C03643=1229.228,50.158,-44.225,-178.947,5.404,148.624
C03644=1229.233,49.908,-44.209,-178.950,5.403,148.624
C03645=1229.238,49.659,-44.193,-178.952,5.403,148.625
C03646=1229.242,49.409,-44.176,-178.955,5.402,148.626
C03647=1229.248,49.160,-44.159,-178.958,5.401,148.626
C03648=1229.253,48.911,-44.143,-178.960,5.401,148.627
C03649=1229.257,48.661,-44.126,-178.962,5.400,148.628
C03650=1229.263,48.412,-44.111,-178.965,5.399,148.628
C03651=1229.267,48.162,-44.094,-178.968,5.399,148.629
C03652=1229.272,47.913,-44.077,-178.970,5.398,148.630
C03653=1229.277,47.664,-44.060,-178.972,5.398,148.630
C03654=1229.282,47.414,-44.044,-178.975,5.398,148.631
C03655=1229.287,47.165,-44.028,-178.978,5.397,148.632
C03656=1229.292,46.915,-44.011,-178.980,5.397,148.632
C03657=1229.296,46.666,-43.995,-178.983,5.396,148.633
C03658=1229.302,46.416,-43.979,-178.986,5.396,148.634
C03659=1229.307,46.167,-43.962,-178.988,5.395,148.634
C03660=1229.312,45.918,-43.946,-178.990,5.394,148.635
C03661=1229.316,45.668,-43.929,-178.993,5.394,148.635
C03662=1229.322,45.419,-43.913,-178.996,5.393,148.636
C03663=1229.326,45.170,-43.897,-178.998,5.392,148.637
C03664=1229.331,44.920,-43.880,-179.000,5.393,148.637
C03665=1229.337,44.670,-43.864,-179.003,5.392,148.638
C03666=1229.341,44.421,-43.847,-179.006,5.392,148.639
C03667=1229.346,44.172,-43.831,-179.008,5.391,148.639
C03668=1229.351,43.922,-43.815,-179.011,5.390,148.640
C03669=1229.356,43.673,-43.799,-179.013,5.389,148.641
C03670=1229.361,43.423,-43.783,-179.016,5.389,148.641
C03671=1229.366,43.174,-43.766,-179.018,5.388,148.642
C03672=1229.371,42.925,-43.750,-179.021,5.388,148.643
C03673=1229.376,42.675,-43.734,-179.023,5.388,148.643
C03674=1229.380,42.426,-43.717,-179.026,5.387,148.644
C03675=1229.386,42.177,-43.702,-179.028,5.387,148.645
C03676=1229.390,41.927,-43.685,-179.031,5.386,148.645
C03677=1229.395,41.678,-43.669,-179.034,5.386,148.646
C03678=1229.401,41.428,-43.652,-179.036,5.385,148.647
C03679=1229.406,41.179,-43.636,-179.039,5.385,148.647
C03680=1229.411,40.929,-43.620,-179.041,5.384,148.648
C03681=1229.416,40.680,-43.604,-179.043,5.384,148.648
C03682=1229.421,40.430,-43.588,-179.046,5.383,148.649
C03683=1229.426,40.181,-43.572,-179.048,5.383,148.650
C03684=1229.430,39.931,-43.556,-179.051,5.382,148.650
C03685=1229.436,39.682,-43.539,-179.054,5.382,148.651
C03686=1229.440,39.432,-43.523,-179.056,5.381,148.652
C03687=1229.445,39.184,-43.507,-179.059,5.381,148.652
C03688=1229.450,38.933,-43.491,-179.062,5.380,148.653
C03689=1229.455,38.685,-43.475,-179.064,5.380,148.654
C03690=1229.460,38.435,-43.459,-179.066,5.380,148.654
C03691=1229.465,38.186,-43.442,-179.069,5.379,148.655
C03692=1229.470,37.936,-43.427,-179.072,5.379,148.656
C03693=1229.475,37.686,-43.411,-179.074,5.378,148.656
C03694=1229.480,37.438,-43.395,-179.076,5.377,148.657
C03695=1229.484,37.188,-43.379,-179.079,5.377,148.658
C03696=1229.490,36.939,-43.363,-179.082,5.376,148.658
C03697=1229.494,36.689,-43.347,-179.084,5.376,148.659
C03698=1229.500,36.439,-43.331,-179.086,5.376,148.660
C03699=1229.504,36.190,-43.315,-179.089,5.375,148.660
C03700=1229.510,35.941,-43.299,-179.092,5.375,148.661
C03701=1229.515,35.692,-43.283,-179.094,5.374,148.662
C03702=1229.519,35.442,-43.267,-179.097,5.374,148.662
C03703=1229.525,35.192,-43.251,-179.100,5.373,148.663
C03704=1229.529,34.943,-43.235,-179.102,5.373,148.664
C03705=1229.535,34.693,-43.219,-179.104,5.373,148.664
C03706=1229.539,34.444,-43.204,-179.107,5.372,148.665
C03707=1229.544,34.195,-43.187,-179.110,5.372,148.666
C03708=1229.549,33.945,-43.172,-179.112,5.371,148.666
C03709=1229.554,33.695,-43.156,-179.114,5.370,148.667
C03710=1229.559,33.446,-43.140,-179.117,5.370,148.668
C03711=1229.564,33.197,-43.124,-179.119,5.370,148.668
C03712=1229.569,32.947,-43.108,-179.122,5.369,148.669
C03713=1229.574,32.698,-43.093,-179.124,5.369,148.670
C03714=1229.578,32.448,-43.076,-179.127,5.368,148.670
C03715=1229.584,32.199,-43.061,-179.130,5.368,148.671
C03716=1229.589,31.950,-43.045,-179.132,5.367,148.672
C03717=1229.594,31.700,-43.029,-179.134,5.367,148.672
C03718=1229.599,31.451,-43.013,-179.137,5.367,148.673
C03719=1229.604,31.202,-42.998,-179.140,5.366,148.674
C03720=1229.608,30.952,-42.982,-179.142,5.366,148.674
C03721=1229.614,30.702,-42.966,-179.145,5.365,148.675
C03722=1229.619,30.453,-42.951,-179.148,5.365,148.676
C03723=1229.624,30.203,-42.934,-179.150,5.365,148.676
C03724=1229.629,29.934,-42.918,-179.152,5.364,148.677
C03725=1229.634,29.666,-42.901,-179.155,5.364,148.678
C03726=1229.640,29.398,-42.884,-179.158,5.363,148.678
C03727=1229.646,29.129,-42.867,-179.160,5.363,148.679
C03728=1229.650,28.879,-42.851,-179.163,5.362,148.680
C03729=1229.655,28.630,-42.836,-179.165,5.361,148.680
C03730=1229.660,28.381,-42.820,-179.168,5.361,148.681
C03731=1229.665,28.131,-42.804,-179.171,5.360,148.682
C03732=1229.670,27.882,-42.789,-179.173,5.361,148.682
C03733=1229.675,27.632,-42.774,-179.175,5.360,148.683
C03734=1229.680,27.382,-42.758,-179.178,5.360,148.684
C03735=1229.685,27.133,-42.742,-179.181,5.359,148.685
C03736=1229.690,26.884,-42.727,-179.183,5.358,148.685
C03737=1229.695,26.634,-42.711,-179.186,5.358,148.686
C03738=1229.700,26.384,-42.696,-179.188,5.358,148.687
C03739=1229.705,26.135,-42.680,-179.191,5.358,148.687
C03740=1229.710,25.886,-42.665,-179.193,5.357,148.688
C03741=1229.715,25.636,-42.649,-179.196,5.357,148.689
C03742=1229.720,25.387,-42.633,-179.199,5.356,148.689
C03743=1229.724,25.138,-42.618,-179.201,5.356,148.690
C03744=1229.730,24.888,-42.602,-179.203,5.356,148.691
C03745=1229.735,24.638,-42.586,-179.206,5.355,148.691
C03746=1229.739,24.389,-42.571,-179.208,5.354,148.692
C03747=1229.745,24.140,-42.556,-179.211,5.354,148.692
C03748=1229.750,23.890,-42.540,-179.214,5.353,148.693
C03749=1229.754,23.641,-42.525,-179.216,5.353,148.694
C03750=1229.760,23.391,-42.510,-179.218,5.353,148.694
C03751=1229.764,23.142,-42.495,-179.221,5.352,148.695
C03752=1229.770,22.892,-42.479,-179.224,5.352,148.696
C03753=1229.775,22.642,-42.463,-179.226,5.351,148.697
C03754=1229.779,22.393,-42.448,-179.228,5.351,148.697
C03755=1229.785,22.144,-42.433,-179.231,5.351,148.698
C03756=1229.790,21.894,-42.417,-179.234,5.350,148.699
C03757=1229.795,21.645,-42.402,-179.236,5.350,148.699
C03758=1229.799,21.395,-42.386,-179.239,5.349,148.700
C03759=1229.804,21.146,-42.371,-179.241,5.350,148.701
C03760=1229.809,20.896,-42.356,-179.244,5.349,148.701
C03761=1229.814,20.647,-42.341,-179.246,5.348,148.702
C03762=1229.819,20.398,-42.325,-179.249,5.348,148.703
C03763=1229.825,20.147,-42.310,-179.251,5.347,148.703
C03764=1229.829,19.898,-42.295,-179.254,5.348,148.704
C03765=1229.835,19.649,-42.279,-179.256,5.347,148.705
C03766=1229.839,19.400,-42.264,-179.259,5.347,148.705
C03767=1229.845,19.150,-42.249,-179.261,5.346,148.706
C03768=1229.849,18.900,-42.233,-179.264,5.346,148.707
C03769=1229.854,18.650,-42.218,-179.266,5.346,148.707
C03770=1229.859,18.401,-42.203,-179.269,5.345,148.708
C03771=1229.864,18.152,-42.188,-179.272,5.345,148.709
C03772=1229.869,17.903,-42.173,-179.274,5.344,148.709
C03773=1229.874,17.653,-42.157,-179.276,5.344,148.710
C03774=1229.879,17.403,-42.143,-179.279,5.344,148.711
C03775=1229.884,17.154,-42.127,-179.282,5.343,148.712
C03776=1229.889,16.905,-42.112,-179.284,5.343,148.712
C03777=1229.894,16.655,-42.096,-179.287,5.342,148.713
C03778=1229.899,16.405,-42.082,-179.289,5.343,148.714
C03779=1229.905,16.156,-42.066,-179.292,5.342,148.714
C03780=1229.909,15.907,-42.051,-179.294,5.341,148.715
C03781=1229.915,15.658,-42.036,-179.297,5.341,148.716
C03782=1229.919,15.407,-42.021,-179.299,5.341,148.716
C03783=1229.924,15.158,-42.006,-179.301,5.340,148.717
C03784=1229.929,14.909,-41.991,-179.304,5.340,148.717
C03785=1229.934,14.659,-41.976,-179.306,5.339,148.718
C03786=1229.939,14.410,-41.961,-179.309,5.339,148.719
C03787=1229.944,14.160,-41.946,-179.311,5.339,148.720
C03788=1229.950,13.910,-41.931,-179.314,5.338,148.720
C03789=1229.954,13.661,-41.916,-179.316,5.338,148.721
C03790=1229.960,13.412,-41.900,-179.319,5.337,148.722
C03791=1229.964,13.162,-41.886,-179.321,5.338,148.722
C03792=1229.969,12.912,-41.871,-179.324,5.337,148.723
C03793=1229.974,12.663,-41.855,-179.326,5.336,148.724
C03794=1229.979,12.413,-41.841,-179.329,5.336,148.724
C03795=1229.984,12.164,-41.825,-179.331,5.336,148.725
C03796=1229.989,11.915,-41.810,-179.334,5.336,148.726
C03797=1229.994,11.665,-41.796,-179.336,5.335,148.726
C03798=1229.999,11.416,-41.780,-179.339,5.335,148.727
C03799=1230.004,11.166,-41.766,-179.341,5.335,148.728
C03800=1230.009,10.917,-41.751,-179.344,5.334,148.728
C03801=1230.015,10.667,-41.736,-179.346,5.334,148.729
C03802=1230.019,10.418,-41.721,-179.349,5.333,148.730
C03803=1230.024,10.169,-41.706,-179.351,5.334,148.730
C03804=1230.030,9.919,-41.691,-179.354,5.333,148.731
C03805=1230.034,9.670,-41.676,-179.356,5.332,148.732
C03806=1230.039,9.420,-41.662,-179.359,5.332,148.733
C03807=1230.045,9.170,-41.647,-179.362,5.331,148.733
C03808=1230.050,8.921,-41.632,-179.364,5.332,148.734
C03809=1230.054,8.672,-41.617,-179.367,5.331,148.735
C03810=1230.060,8.422,-41.602,-179.369,5.331,148.735
C03811=1230.064,8.172,-41.587,-179.372,5.330,148.736
C03812=1230.069,7.922,-41.573,-179.374,5.330,148.737
C03813=1230.074,7.673,-41.558,-179.377,5.330,148.737
C03814=1230.079,7.423,-41.543,-179.379,5.329,148.738
C03815=1230.084,7.174,-41.528,-179.381,5.330,148.739
C03816=1230.089,6.924,-41.514,-179.384,5.329,148.739
C03817=1230.094,6.675,-41.499,-179.387,5.329,148.740
C03818=1230.099,6.425,-41.484,-179.389,5.328,148.741
C03819=1230.104,6.175,-41.469,-179.391,5.328,148.741
C03820=1230.109,5.926,-41.455,-179.394,5.328,148.742
C03821=1230.114,5.677,-41.440,-179.397,5.327,148.743
C03822=1230.120,5.428,-41.425,-179.399,5.327,148.744
C03823=1230.125,5.178,-41.411,-179.401,5.327,148.744
C03824=1230.130,4.928,-41.396,-179.404,5.326,148.745
C03825=1230.134,4.679,-41.381,-179.407,5.326,148.746
C03826=1230.140,4.429,-41.367,-179.409,5.325,148.746
C03827=1230.145,4.180,-41.352,-179.411,5.326,148.747
C03828=1230.150,3.911,-41.337,-179.414,5.325,148.748
C03829=1230.155,3.642,-41.321,-179.417,5.325,148.749
C03830=1230.161,3.373,-41.305,-179.420,5.324,148.749
C03831=1230.166,3.104,-41.289,-179.422,5.324,148.750
C03832=1230.171,2.854,-41.275,-179.425,5.323,148.751
C03833=1230.176,2.605,-41.260,-179.427,5.324,148.751
C03834=1230.181,2.356,-41.245,-179.430,5.323,148.752
C03835=1230.187,2.106,-41.230,-179.432,5.323,148.753
C03836=1230.191,1.857,-41.215,-179.435,5.323,148.753
C03837=1230.196,1.607,-41.201,-179.437,5.322,148.754
C03838=1230.201,1.357,-41.187,-179.440,5.322,148.755
C03839=1230.207,1.108,-41.173,-179.443,5.321,148.755
C03840=1230.211,0.859,-41.158,-179.445,5.322,148.756
C03841=1230.216,0.609,-41.144,-179.447,5.321,148.757
C03842=1230.222,0.359,-41.129,-179.450,5.321,148.758
C03843=1230.227,0.110,-41.115,-179.453,5.320,148.758
C03844=1230.232,-0.139,-41.100,-179.455,5.320,148.759
C03845=1230.237,-0.389,-41.085,-179.457,5.320,148.760
C03846=1230.241,-0.639,-41.071,-179.460,5.319,148.760
C03847=1230.246,-0.889,-41.057,-179.462,5.320,148.761
C03848=1230.252,-1.138,-41.043,-179.465,5.319,148.762
C03849=1230.257,-1.387,-41.028,-179.467,5.318,148.762
C03850=1230.262,-1.636,-41.014,-179.470,5.318,148.763
C03851=1230.267,-1.886,-40.999,-179.472,5.318,148.764
C03852=1230.272,-2.136,-40.985,-179.475,5.318,148.764
C03853=1230.276,-2.386,-40.971,-179.477,5.317,148.765
C03854=1230.282,-2.636,-40.956,-179.479,5.317,148.766
C03855=1230.287,-2.885,-40.941,-179.482,5.317,148.766
C03856=1230.292,-3.134,-40.927,-179.485,5.317,148.767
C03857=1230.297,-3.383,-40.913,-179.487,5.317,148.768
C03858=1230.302,-3.633,-40.898,-179.490,5.317,148.769
C03859=1230.307,-3.883,-40.884,-179.493,5.316,148.769
C03860=1230.312,-4.133,-40.870,-179.495,5.316,148.770
C03861=1230.317,-4.382,-40.856,-179.497,5.316,148.771
C03862=1230.323,-4.631,-40.842,-179.500,5.315,148.772
C03863=1230.327,-4.880,-40.827,-179.503,5.315,148.772
C03864=1230.332,-5.130,-40.812,-179.505,5.315,148.773
C03865=1230.337,-5.380,-40.798,-179.507,5.315,148.774
C03866=1230.342,-5.629,-40.784,-179.510,5.314,148.774
C03867=1230.347,-5.879,-40.770,-179.513,5.313,148.775
C03868=1230.353,-6.128,-40.756,-179.515,5.314,148.776
C03869=1230.358,-6.378,-40.741,-179.517,5.313,148.776
C03870=1230.363,-6.628,-40.727,-179.520,5.313,148.777
C03871=1230.368,-6.877,-40.713,-179.522,5.313,148.778
C03872=1230.373,-7.127,-40.699,-179.525,5.312,148.778
C03873=1230.378,-7.376,-40.685,-179.528,5.312,148.779
C03874=1230.382,-7.625,-40.671,-179.530,5.312,148.780
C03875=1230.387,-7.875,-40.657,-179.532,5.312,148.781
C03876=1230.392,-8.125,-40.642,-179.535,5.311,148.781
C03877=1230.397,-8.375,-40.628,-179.537,5.312,148.782
C03878=1230.403,-8.624,-40.614,-179.540,5.311,148.783
C03879=1230.408,-8.873,-40.600,-179.542,5.310,148.783
C03880=1230.413,-9.123,-40.586,-179.545,5.310,148.784
C03881=1230.418,-9.373,-40.571,-179.547,5.310,148.785
C03882=1230.423,-9.622,-40.557,-179.550,5.310,148.785
C03883=1230.428,-9.871,-40.543,-179.552,5.309,148.786
C03884=1230.433,-10.121,-40.529,-179.554,5.309,148.787
C03885=1230.438,-10.371,-40.515,-179.557,5.309,148.787
C03886=1230.443,-10.620,-40.502,-179.560,5.308,148.788
C03887=1230.448,-10.870,-40.488,-179.562,5.309,148.789
C03888=1230.453,-11.120,-40.473,-179.564,5.308,148.790
C03889=1230.458,-11.369,-40.459,-179.567,5.308,148.790
C03890=1230.464,-11.618,-40.445,-179.569,5.308,148.791
C03891=1230.469,-11.868,-40.431,-179.572,5.307,148.792
C03892=1230.473,-12.118,-40.417,-179.575,5.307,148.792
C03893=1230.478,-12.367,-40.403,-179.577,5.307,148.793
C03894=1230.484,-12.617,-40.390,-179.579,5.307,148.794
C03895=1230.489,-12.866,-40.376,-179.582,5.306,148.794
C03896=1230.493,-13.116,-40.361,-179.584,5.307,148.795
C03897=1230.499,-13.365,-40.347,-179.587,5.306,148.796
C03898=1230.504,-13.615,-40.333,-179.589,5.306,148.796
C03899=1230.508,-13.864,-40.319,-179.591,5.306,148.797
C03900=1230.513,-14.115,-40.306,-179.595,5.306,148.798
C03901=1230.519,-14.364,-40.292,-179.597,5.305,148.799
C03902=1230.524,-14.613,-40.278,-179.599,5.305,148.799
C03903=1230.529,-14.863,-40.263,-179.602,5.305,148.800
C03904=1230.534,-15.112,-40.251,-179.605,5.304,148.801
C03905=1230.539,-15.362,-40.237,-179.607,5.305,148.802
C03906=1230.544,-15.612,-40.222,-179.609,5.304,148.802
C03907=1230.550,-15.861,-40.208,-179.612,5.304,148.803
C03908=1230.554,-16.111,-40.195,-179.614,5.304,148.804
C03909=1230.559,-16.361,-40.181,-179.617,5.303,148.804
C03910=1230.565,-16.610,-40.167,-179.619,5.303,148.805
C03911=1230.569,-16.859,-40.153,-179.621,5.303,148.806
C03912=1230.574,-17.109,-40.140,-179.624,5.303,148.806
C03913=1230.580,-17.358,-40.126,-179.627,5.302,148.807
C03914=1230.585,-17.608,-40.112,-179.629,5.303,148.808
C03915=1230.590,-17.858,-40.098,-179.632,5.302,148.808
C03916=1230.595,-18.107,-40.085,-179.634,5.302,148.809
C03917=1230.600,-18.357,-40.071,-179.636,5.302,148.810
C03918=1230.605,-18.607,-40.057,-179.639,5.301,148.811
C03919=1230.610,-18.856,-40.043,-179.642,5.301,148.811
C03920=1230.615,-19.105,-40.029,-179.644,5.301,148.812
C03921=1230.620,-19.355,-40.016,-179.646,5.301,148.813
C03922=1230.625,-19.605,-40.002,-179.649,5.300,148.813
C03923=1230.630,-19.854,-39.988,-179.651,5.300,148.814
C03924=1230.635,-20.104,-39.975,-179.654,5.300,148.815
C03925=1230.640,-20.354,-39.961,-179.656,5.299,148.815
C03926=1230.645,-20.602,-39.948,-179.658,5.300,148.816
C03927=1230.651,-20.853,-39.934,-179.661,5.299,148.817
C03928=1230.655,-21.102,-39.920,-179.664,5.299,148.818
C03929=1230.661,-21.352,-39.907,-179.666,5.299,148.818
C03930=1230.666,-21.601,-39.893,-179.669,5.299,148.819
C03931=1230.671,-21.851,-39.880,-179.672,5.298,148.820
C03932=1230.676,-22.120,-39.865,-179.674,5.299,148.821
C03933=1230.682,-22.389,-39.850,-179.676,5.298,148.821
C03934=1230.687,-22.659,-39.835,-179.679,5.298,148.822
C03935=1230.693,-22.928,-39.821,-179.682,5.297,148.823
C03936=1230.698,-23.178,-39.808,-179.684,5.298,148.824
C03937=1230.702,-23.427,-39.793,-179.687,5.297,148.824
C03938=1230.708,-23.677,-39.780,-179.690,5.297,148.825
C03939=1230.713,-23.926,-39.766,-179.692,5.297,148.826
C03940=1230.718,-24.176,-39.753,-179.694,5.297,148.826
C03941=1230.723,-24.425,-39.740,-179.696,5.297,148.827
C03942=1230.729,-24.675,-39.726,-179.699,5.296,148.828
C03943=1230.733,-24.924,-39.713,-179.702,5.296,148.828
C03944=1230.738,-25.175,-39.699,-179.704,5.296,148.829
C03945=1230.744,-25.424,-39.685,-179.706,5.296,148.830
C03946=1230.748,-25.674,-39.672,-179.709,5.295,148.831
C03947=1230.754,-25.923,-39.658,-179.711,5.295,148.831
C03948=1230.758,-26.173,-39.645,-179.714,5.295,148.832
C03949=1230.764,-26.422,-39.631,-179.717,5.294,148.833
C03950=1230.768,-26.672,-39.619,-179.719,5.295,148.833
C03951=1230.774,-26.921,-39.605,-179.721,5.294,148.834
C03952=1230.778,-27.171,-39.592,-179.723,5.295,148.835
C03953=1230.784,-27.420,-39.578,-179.726,5.294,148.835
C03954=1230.788,-27.670,-39.565,-179.729,5.293,148.836
C03955=1230.794,-27.920,-39.552,-179.731,5.294,148.837
C03956=1230.799,-28.170,-39.539,-179.733,5.293,148.837
C03957=1230.804,-28.419,-39.525,-179.736,5.293,148.838
C03958=1230.809,-28.669,-39.512,-179.739,5.293,148.839
C03959=1230.815,-28.918,-39.499,-179.741,5.293,148.840
C03960=1230.819,-29.168,-39.485,-179.743,5.293,148.841
C03961=1230.825,-29.417,-39.472,-179.746,5.293,148.841
C03962=1230.829,-29.667,-39.458,-179.749,5.292,148.842
C03963=1230.835,-29.916,-39.445,-179.751,5.293,148.843
C03964=1230.839,-30.166,-39.432,-179.753,5.292,148.843
C03965=1230.845,-30.416,-39.419,-179.756,5.292,148.844
C03966=1230.849,-30.665,-39.405,-179.758,5.292,148.845
C03967=1230.855,-30.915,-39.392,-179.761,5.291,148.845
C03968=1230.860,-31.165,-39.379,-179.763,5.292,148.846
C03969=1230.865,-31.414,-39.365,-179.766,5.291,148.847
C03970=1230.871,-31.663,-39.352,-179.768,5.291,148.847
C03971=1230.875,-31.913,-39.339,-179.770,5.291,148.848
C03972=1230.881,-32.163,-39.326,-179.773,5.291,148.849
C03973=1230.885,-32.412,-39.312,-179.776,5.290,148.850
C03974=1230.891,-32.662,-39.299,-179.778,5.290,148.850
C03975=1230.896,-32.912,-39.286,-179.780,5.290,148.851
C03976=1230.901,-33.161,-39.274,-179.783,5.290,148.852
C03977=1230.906,-33.411,-39.259,-179.785,5.290,148.852
C03978=1230.911,-33.660,-39.247,-179.788,5.289,148.853
C03979=1230.917,-33.910,-39.234,-179.790,5.289,148.854
C03980=1230.921,-34.160,-39.221,-179.793,5.289,148.854
C03981=1230.926,-34.409,-39.208,-179.795,5.289,148.855
C03982=1230.931,-34.659,-39.194,-179.797,5.289,148.856
C03983=1230.936,-34.908,-39.181,-179.801,5.289,148.857
C03984=1230.942,-35.158,-39.168,-179.803,5.289,148.858
C03985=1230.947,-35.408,-39.155,-179.805,5.288,148.858
C03986=1230.952,-35.657,-39.142,-179.807,5.289,148.859
C03987=1230.957,-35.907,-39.128,-179.810,5.288,148.860
C03988=1230.962,-36.156,-39.115,-179.813,5.288,148.860
C03989=1230.967,-36.406,-39.103,-179.815,5.288,148.861
C03990=1230.972,-36.656,-39.089,-179.817,5.288,148.862
C03991=1230.977,-36.905,-39.077,-179.820,5.287,148.862
C03992=1230.983,-37.155,-39.064,-179.822,5.287,148.863
C03993=1230.988,-37.405,-39.051,-179.825,5.287,148.864
C03994=1230.993,-37.654,-39.038,-179.827,5.287,148.865
C03995=1230.997,-37.904,-39.025,-179.830,5.287,148.865
C03996=1231.003,-38.153,-39.011,-179.832,5.286,148.866
C03997=1231.008,-38.403,-38.998,-179.834,5.287,148.867
C03998=1231.013,-38.653,-38.986,-179.837,5.286,148.867
C03999=1231.018,-38.902,-38.973,-179.839,5.286,148.868
C04000=1231.024,-39.152,-38.960,-179.842,5.286,148.869
C04001=1231.028,-39.402,-38.947,-179.844,5.285,148.869
C04002=1231.033,-39.651,-38.934,-179.846,5.286,148.870
C04003=1231.038,-39.900,-38.922,-179.849,5.285,148.871
C04004=1231.044,-40.151,-38.908,-179.851,5.286,148.872
C04005=1231.049,-40.400,-38.895,-179.854,5.285,148.872
C04006=1231.054,-40.649,-38.883,-179.856,5.285,148.873
C04007=1231.058,-40.899,-38.870,-179.859,5.285,148.874
C04008=1231.064,-41.149,-38.857,-179.862,5.285,148.875
C04009=1231.069,-41.398,-38.844,-179.864,5.285,148.875
C04010=1231.074,-41.648,-38.831,-179.867,5.285,148.876
C04011=1231.079,-41.897,-38.818,-179.869,5.285,148.877
C04012=1231.085,-42.147,-38.805,-179.871,5.284,148.877
C04013=1231.089,-42.397,-38.792,-179.874,5.284,148.878
C04014=1231.095,-42.646,-38.780,-179.876,5.284,148.879
C04015=1231.100,-42.896,-38.767,-179.879,5.284,148.879
C04016=1231.105,-43.145,-38.754,-179.881,5.284,148.880
C04017=1231.110,-43.395,-38.741,-179.883,5.284,148.881
C04018=1231.115,-43.645,-38.728,-179.886,5.283,148.882
C04019=1231.120,-43.894,-38.716,-179.888,5.283,148.882
C04020=1231.125,-44.145,-38.703,-179.891,5.283,148.883
C04021=1231.130,-44.394,-38.691,-179.893,5.283,148.884
C04022=1231.135,-44.643,-38.678,-179.896,5.283,148.884
C04023=1231.141,-44.893,-38.665,-179.898,5.283,148.885
C04024=1231.146,-45.143,-38.652,-179.900,5.283,148.886
C04025=1231.151,-45.392,-38.640,-179.903,5.282,148.886
C04026=1231.156,-45.642,-38.627,-179.905,5.282,148.887
C04027=1231.161,-45.891,-38.614,-179.908,5.282,148.888
C04028=1231.166,-46.142,-38.602,-179.910,5.282,148.889
C04029=1231.171,-46.391,-38.589,-179.913,5.282,148.889
C04030=1231.177,-46.640,-38.576,-179.915,5.281,148.890
C04031=1231.182,-46.890,-38.564,-179.917,5.282,148.891
C04032=1231.187,-47.140,-38.551,-179.920,5.281,148.892
C04033=1231.192,-47.389,-38.538,-179.923,5.282,148.892
C04034=1231.197,-47.639,-38.526,-179.925,5.281,148.893
C04035=1231.202,-47.888,-38.514,-179.927,5.282,148.894
C04036=1231.207,-48.158,-38.500,-179.930,5.281,148.894
C04037=1231.213,-48.428,-38.486,-179.933,5.281,148.895
C04038=1231.219,-48.697,-38.472,-179.935,5.280,148.896
C04039=1231.224,-48.968,-38.459,-179.938,5.281,148.897
C04040=1231.229,-49.217,-38.447,-179.941,5.280,148.897
C04041=1231.235,-49.466,-38.434,-179.943,5.281,148.898
C04042=1231.239,-49.716,-38.421,-179.945,5.280,148.899
C04043=1231.245,-49.966,-38.409,-179.947,5.281,148.900
C04044=1231.250,-50.216,-38.396,-179.950,5.280,148.900
C04045=1231.255,-50.465,-38.384,-179.953,5.280,148.901
C04046=1231.261,-50.715,-38.372,-179.955,5.280,148.902
C04047=1231.265,-50.965,-38.359,-179.957,5.279,148.902
C04048=1231.270,-51.214,-38.346,-179.960,5.280,148.903
C04049=1231.275,-51.464,-38.333,-179.962,5.279,148.904
C04050=1231.281,-51.714,-38.322,-179.964,5.280,148.904
C04051=1231.286,-51.963,-38.309,-179.967,5.279,148.905
C04052=1231.290,-52.213,-38.296,-179.970,5.279,148.906
C04053=1231.296,-52.463,-38.284,-179.972,5.279,148.907
C04054=1231.301,-52.712,-38.272,-179.974,5.278,148.907
C04055=1231.306,-52.961,-38.259,-179.976,5.279,148.908
C04056=1231.312,-53.211,-38.247,-179.979,5.278,148.909
C04057=1231.317,-53.461,-38.234,-179.981,5.279,148.909
C04058=1231.321,-53.711,-38.221,-179.984,5.278,148.910
C04059=1231.327,-53.961,-38.210,-179.987,5.278,148.911
C04060=1231.332,-54.210,-38.197,-179.989,5.278,148.912
C04061=1231.337,-54.460,-38.185,-179.992,5.278,148.912
C04062=1231.342,-54.709,-38.172,-179.994,5.278,148.913
C04063=1231.347,-54.958,-38.160,-179.997,5.278,148.914
C04064=1231.352,-55.208,-38.149,-179.999,5.278,148.915
C04065=1231.357,-55.458,-38.136,179.999,5.278,148.915
C04066=1231.362,-55.708,-38.124,179.997,5.278,148.916
C04067=1231.367,-55.957,-38.111,179.994,5.277,148.917
C04068=1231.372,-56.207,-38.099,179.991,5.277,148.917
C04069=1231.378,-56.457,-38.087,179.989,5.277,148.918
C04070=1231.383,-56.706,-38.074,179.987,5.277,148.919
C04071=1231.388,-56.956,-38.062,179.984,5.277,148.920
C04072=1231.393,-57.205,-38.050,179.982,5.277,148.920
C04073=1231.399,-57.455,-38.038,179.980,5.277,148.921
C04074=1231.403,-57.705,-38.025,179.977,5.276,148.922
C04075=1231.408,-57.955,-38.013,179.975,5.277,148.922
C04076=1231.413,-58.204,-38.001,179.972,5.276,148.923
C04077=1231.419,-58.454,-37.989,179.970,5.277,148.924
C04078=1231.424,-58.703,-37.976,179.967,5.276,148.924
C04079=1231.429,-58.953,-37.964,179.965,5.276,148.925
C04080=1231.434,-59.203,-37.952,179.963,5.276,148.926
C04081=1231.440,-59.453,-37.940,179.960,5.276,148.927
C04082=1231.444,-59.702,-37.928,179.958,5.276,148.927
C04083=1231.449,-59.952,-37.916,179.955,5.275,148.928
C04084=1231.455,-60.201,-37.903,179.953,5.276,148.929
C04085=1231.460,-60.451,-37.892,179.951,5.275,148.929
C04086=1231.465,-60.701,-37.880,179.948,5.276,148.930
C04087=1231.470,-60.951,-37.867,179.946,5.275,148.931
C04088=1231.475,-61.200,-37.855,179.944,5.275,148.931
C04089=1231.480,-61.450,-37.843,179.941,5.275,148.932
C04090=1231.485,-61.700,-37.831,179.938,5.275,148.933
C04091=1231.490,-61.949,-37.818,179.936,5.275,148.934
C04092=1231.496,-62.199,-37.806,179.933,5.275,148.935
C04093=1231.500,-62.449,-37.795,179.931,5.275,148.935
C04094=1231.506,-62.698,-37.783,179.928,5.275,148.936
C04095=1231.511,-62.948,-37.771,179.926,5.275,148.937
C04096=1231.516,-63.198,-37.759,179.924,5.274,148.937
C04097=1231.522,-63.447,-37.746,179.922,5.275,148.938
C04098=1231.526,-63.697,-37.735,179.919,5.274,148.939
C04099=1231.532,-63.947,-37.723,179.917,5.275,148.939
C04100=1231.537,-64.196,-37.710,179.914,5.274,148.940
C04101=1231.542,-64.446,-37.699,179.912,5.275,148.941
C04102=1231.547,-64.696,-37.687,179.909,5.274,148.942
C04103=1231.552,-64.945,-37.675,179.907,5.274,148.942
C04104=1231.558,-65.195,-37.663,179.905,5.274,148.943
C04105=1231.563,-65.445,-37.651,179.902,5.273,148.944
C04106=1231.567,-65.694,-37.639,179.900,5.274,148.944
C04107=1231.573,-65.944,-37.627,179.897,5.273,148.945
C04108=1231.578,-66.194,-37.615,179.895,5.274,148.946
C04109=1231.583,-66.443,-37.603,179.892,5.273,148.947
C04110=1231.588,-66.693,-37.591,179.890,5.273,148.947
C04111=1231.593,-66.942,-37.579,179.888,5.273,148.948
C04112=1231.599,-67.192,-37.567,179.886,5.273,148.949
C04113=1231.603,-67.441,-37.555,179.883,5.273,148.949
C04114=1231.609,-67.691,-37.544,179.881,5.273,148.950
C04115=1231.614,-67.941,-37.532,179.878,5.273,148.951
C04116=1231.619,-68.191,-37.520,179.876,5.273,148.952
C04117=1231.625,-68.440,-37.509,179.873,5.273,148.952
C04118=1231.630,-68.689,-37.496,179.871,5.273,148.953
C04119=1231.635,-68.939,-37.485,179.869,5.272,148.954
C04120=1231.640,-69.189,-37.473,179.866,5.272,148.954
C04121=1231.646,-69.439,-37.461,179.864,5.272,148.955
C04122=1231.650,-69.689,-37.450,179.861,5.272,148.956
C04123=1231.655,-69.938,-37.437,179.859,5.272,148.956
C04124=1231.661,-70.188,-37.425,179.856,5.272,148.957
C04125=1231.665,-70.437,-37.414,179.854,5.272,148.958
C04126=1231.671,-70.687,-37.402,179.852,5.272,148.959
C04127=1231.676,-70.937,-37.391,179.850,5.272,148.959
C04128=1231.681,-71.187,-37.379,179.847,5.272,148.960
C04129=1231.686,-71.437,-37.367,179.845,5.272,148.961
C04130=1231.691,-71.685,-37.356,179.842,5.271,148.961
C04131=1231.697,-71.935,-37.344,179.840,5.272,148.962
C04132=1231.702,-72.185,-37.332,179.837,5.271,148.963
C04133=1231.707,-72.435,-37.321,179.835,5.272,148.964
C04134=1231.712,-72.685,-37.309,179.833,5.271,148.964
C04135=1231.717,-72.934,-37.297,179.831,5.271,148.965
C04136=1231.723,-73.184,-37.285,179.827,5.271,148.966
C04137=1231.728,-73.434,-37.274,179.825,5.272,148.967
C04138=1231.733,-73.684,-37.262,179.823,5.271,148.967
C04139=1231.739,-73.933,-37.251,179.821,5.272,148.968
C04140=1231.744,-74.203,-37.238,179.818,5.271,148.969
C04141=1231.749,-74.474,-37.225,179.815,5.271,148.969
C04142=1231.756,-74.744,-37.213,179.813,5.271,148.970
C04143=1231.760,-75.014,-37.201,179.810,5.271,148.971
C04144=1231.766,-75.264,-37.189,179.807,5.270,148.972
C04145=1231.771,-75.514,-37.177,179.805,5.271,148.973
C04146=1231.776,-75.763,-37.166,179.802,5.270,148.973
C04147=1231.782,-76.013,-37.154,179.800,5.271,148.974
C04148=1231.786,-76.262,-37.143,179.798,5.270,148.975
C04149=1231.792,-76.512,-37.131,179.796,5.271,148.975
C04150=1231.796,-76.762,-37.120,179.793,5.270,148.976
C04151=1231.802,-77.012,-37.108,179.791,5.270,148.977
C04152=1231.807,-77.261,-37.097,179.788,5.270,148.977
C04153=1231.813,-77.511,-37.085,179.786,5.270,148.978
C04154=1231.817,-77.760,-37.074,179.783,5.270,148.979
C04155=1231.823,-78.010,-37.062,179.781,5.270,148.980
C04156=1231.827,-78.260,-37.050,179.779,5.270,148.980
C04157=1231.833,-78.510,-37.038,179.777,5.270,148.981
C04158=1231.838,-78.759,-37.028,179.774,5.270,148.982
C04159=1231.844,-79.009,-37.016,179.772,5.270,148.982
C04160=1231.849,-79.259,-37.005,179.769,5.270,148.983
C04161=1231.853,-79.509,-36.994,179.767,5.270,148.984
C04162=1231.859,-79.759,-36.982,179.764,5.269,148.985
C04163=1231.864,-80.007,-36.971,179.762,5.270,148.985
C04164=1231.869,-80.257,-36.959,179.760,5.269,148.986
C04165=1231.874,-80.507,-36.948,179.758,5.270,148.987
C04166=1231.880,-80.757,-36.936,179.755,5.269,148.987
C04167=1231.884,-81.007,-36.925,179.753,5.270,148.988
C04168=1231.890,-81.256,-36.914,179.750,5.269,148.989
C04169=1231.895,-81.506,-36.903,179.748,5.269,148.990
C04170=1231.900,-81.756,-36.891,179.745,5.269,148.990
C04171=1231.905,-82.006,-36.879,179.743,5.269,148.991
C04172=1231.911,-82.255,-36.868,179.741,5.269,148.992
C04173=1231.915,-82.504,-36.857,179.738,5.269,148.992
C04174=1231.921,-82.755,-36.846,179.736,5.269,148.993
C04175=1231.926,-83.004,-36.835,179.734,5.269,148.994
C04176=1231.932,-83.254,-36.823,179.731,5.269,148.994
C04177=1231.937,-83.503,-36.812,179.729,5.269,148.995
C04178=1231.941,-83.753,-36.801,179.726,5.269,148.996
C04179=1231.947,-84.003,-36.789,179.724,5.269,148.997
C04180=1231.952,-84.252,-36.779,179.722,5.268,148.997
C04181=1231.957,-84.502,-36.767,179.719,5.269,148.998
C04182=1231.962,-84.752,-36.755,179.717,5.268,148.999
C04183=1231.967,-85.002,-36.745,179.715,5.269,148.999
C04184=1231.973,-85.251,-36.734,179.712,5.268,149.000
C04185=1231.978,-85.501,-36.722,179.710,5.269,149.001
C04186=1231.983,-85.751,-36.711,179.707,5.268,149.002
C04187=1231.988,-86.001,-36.700,179.705,5.268,149.002
C04188=1231.994,-86.250,-36.689,179.702,5.268,149.003
C04189=1231.998,-86.500,-36.677,179.700,5.268,149.004
C04190=1232.003,-86.749,-36.666,179.698,5.268,149.004
C04191=1232.010,-86.999,-36.655,179.696,5.268,149.005
C04192=1232.014,-87.249,-36.644,179.693,5.268,149.006
C04193=1232.019,-87.498,-36.633,179.691,5.268,149.007
C04194=1232.025,-87.748,-36.622,179.688,5.268,149.007
C04195=1232.030,-87.998,-36.611,179.686,5.268,149.008
C04196=1232.035,-88.248,-36.599,179.683,5.268,149.009
C04197=1232.040,-88.498,-36.589,179.682,5.268,149.009
C04198=1232.045,-88.747,-36.578,179.679,5.267,149.010
C04199=1232.050,-88.997,-36.566,179.677,5.267,149.011
C04200=1232.055,-89.247,-36.555,179.674,5.267,149.011
C04201=1232.061,-89.496,-36.544,179.672,5.267,149.012
C04202=1232.066,-89.746,-36.534,179.670,5.268,149.013
C04203=1232.071,-89.996,-36.522,179.668,5.267,149.013
C04204=1232.076,-90.245,-36.511,179.665,5.268,149.014
C04205=1232.081,-90.495,-36.500,179.663,5.267,149.015
C04206=1232.086,-90.745,-36.489,179.661,5.267,149.016
C04207=1232.092,-90.995,-36.478,179.658,5.267,149.016
C04208=1232.097,-91.244,-36.467,179.656,5.267,149.017
C04209=1232.102,-91.493,-36.456,179.653,5.267,149.018
C04210=1232.107,-91.743,-36.445,179.651,5.267,149.018
C04211=1232.112,-91.993,-36.434,179.648,5.267,149.019
C04212=1232.118,-92.243,-36.423,179.646,5.267,149.020
C04213=1232.123,-92.493,-36.412,179.644,5.267,149.021
C04214=1232.128,-92.743,-36.402,179.642,5.267,149.021
C04215=1232.133,-92.992,-36.391,179.639,5.267,149.022
C04216=1232.138,-93.242,-36.380,179.637,5.267,149.023
C04217=1232.144,-93.491,-36.369,179.634,5.267,149.023
C04218=1232.149,-93.741,-36.358,179.632,5.267,149.024
C04219=1232.154,-93.991,-36.347,179.629,5.266,149.025
C04220=1232.160,-94.241,-36.336,179.627,5.267,149.026
C04221=1232.164,-94.490,-36.325,179.625,5.266,149.026
C04222=1232.170,-94.740,-36.315,179.623,5.267,149.027
C04223=1232.175,-94.990,-36.303,179.620,5.266,149.028
C04224=1232.180,-95.240,-36.292,179.618,5.267,149.028
C04225=1232.186,-95.489,-36.282,179.615,5.266,149.029
C04226=1232.191,-95.739,-36.271,179.613,5.267,149.030
C04227=1232.196,-95.988,-36.260,179.610,5.266,149.031
C04228=1232.201,-96.238,-36.249,179.608,5.266,149.031
C04229=1232.206,-96.488,-36.238,179.606,5.267,149.032
C04230=1232.211,-96.737,-36.228,179.603,5.266,149.033
C04231=1232.217,-96.988,-36.217,179.601,5.267,149.033
C04232=1232.222,-97.237,-36.206,179.599,5.266,149.034
C04233=1232.227,-97.487,-36.195,179.597,5.267,149.035
C04234=1232.233,-97.736,-36.184,179.594,5.266,149.036
C04235=1232.238,-97.986,-36.174,179.592,5.266,149.036
C04236=1232.243,-98.236,-36.164,179.590,5.266,149.037
C04237=1232.248,-98.486,-36.152,179.588,5.266,149.037
C04238=1232.253,-98.736,-36.142,179.585,5.266,149.038
C04239=1232.258,-98.985,-36.131,179.583,5.266,149.039
C04240=1232.263,-99.235,-36.120,179.580,5.266,149.040
C04241=1232.269,-99.485,-36.110,179.578,5.266,149.040
C04242=1232.273,-99.734,-36.099,179.575,5.265,149.041
C04243=1232.279,-99.984,-36.089,179.573,5.266,149.042
C04244=1232.285,-100.255,-36.076,179.571,5.265,149.042
C04245=1232.291,-100.526,-36.065,179.568,5.266,149.043
C04246=1232.296,-100.796,-36.053,179.565,5.266,149.044
C04247=1232.302,-101.068,-36.042,179.563,5.266,149.045
C04248=1232.307,-101.318,-36.031,179.561,5.266,149.046
C04249=1232.312,-101.567,-36.020,179.558,5.266,149.046
C04250=1232.317,-101.817,-36.010,179.556,5.266,149.047
C04251=1232.323,-102.067,-36.000,179.554,5.266,149.048
C04252=1232.328,-102.316,-35.988,179.551,5.265,149.048
C04253=1232.333,-102.566,-35.978,179.549,5.266,149.049
C04254=1232.338,-102.816,-35.968,179.546,5.265,149.050
C04255=1232.344,-103.066,-35.957,179.544,5.266,149.051
C04256=1232.348,-103.315,-35.946,179.541,5.265,149.051
C04257=1232.354,-103.565,-35.936,179.540,5.265,149.052
C04258=1232.359,-103.815,-35.925,179.537,5.265,149.052
C04259=1232.365,-104.065,-35.915,179.535,5.265,149.053
C04260=1232.370,-104.314,-35.904,179.532,5.265,149.054
C04261=1232.374,-104.564,-35.894,179.530,5.265,149.055
C04262=1232.380,-104.813,-35.884,179.528,5.265,149.055
C04263=1232.385,-105.063,-35.873,179.526,5.265,149.056
C04264=1232.390,-105.313,-35.863,179.523,5.265,149.057
C04265=1232.395,-105.563,-35.852,179.521,5.265,149.057
C04266=1232.401,-105.812,-35.842,179.519,5.265,149.058
C04267=1232.406,-106.062,-35.831,179.516,5.265,149.059
C04268=1232.411,-106.312,-35.821,179.514,5.265,149.060
C04269=1232.416,-106.562,-35.810,179.511,5.265,149.060
C04270=1232.422,-106.812,-35.800,179.509,5.265,149.061
C04271=1232.427,-107.061,-35.789,179.506,5.265,149.062
C04272=1232.432,-107.311,-35.779,179.504,5.265,149.062
C04273=1232.438,-107.560,-35.768,179.502,5.264,149.063
C04274=1232.442,-107.810,-35.758,179.500,5.265,149.064
C04275=1232.448,-108.060,-35.748,179.497,5.264,149.064
C04276=1232.453,-108.310,-35.738,179.495,5.265,149.065
C04277=1232.458,-108.560,-35.727,179.493,5.265,149.066
C04278=1232.464,-108.809,-35.717,179.491,5.264,149.066
C04279=1232.469,-109.059,-35.706,179.488,5.265,149.067
C04280=1232.474,-109.308,-35.696,179.486,5.264,149.068
C04281=1232.479,-109.559,-35.685,179.484,5.265,149.069
C04282=1232.484,-109.808,-35.676,179.481,5.264,149.069
C04283=1232.490,-110.057,-35.665,179.479,5.265,149.070
C04284=1232.495,-110.308,-35.655,179.476,5.264,149.071
C04285=1232.500,-110.557,-35.645,179.474,5.265,149.071
C04286=1232.505,-110.807,-35.634,179.471,5.264,149.072
C04287=1232.511,-111.057,-35.624,179.470,5.264,149.073
C04288=1232.516,-111.306,-35.614,179.468,5.265,149.073
C04289=1232.521,-111.556,-35.604,179.465,5.264,149.074
C04290=1232.526,-111.806,-35.593,179.463,5.264,149.075
C04291=1232.531,-112.056,-35.583,179.460,5.264,149.076
C04292=1232.537,-112.306,-35.573,179.458,5.264,149.076
C04293=1232.542,-112.555,-35.563,179.456,5.264,149.077
C04294=1232.547,-112.805,-35.552,179.453,5.264,149.078
C04295=1232.552,-113.055,-35.542,179.451,5.264,149.078
C04296=1232.558,-113.304,-35.532,179.449,5.264,149.079
C04297=1232.563,-113.555,-35.521,179.446,5.264,149.080
C04298=1232.568,-113.804,-35.512,179.444,5.264,149.081
C04299=1232.573,-114.053,-35.502,179.442,5.264,149.081
C04300=1232.578,-114.304,-35.491,179.440,5.264,149.082
C04301=1232.584,-114.553,-35.481,179.438,5.264,149.082
C04302=1232.589,-114.802,-35.471,179.435,5.264,149.083
C04303=1232.594,-115.053,-35.461,179.433,5.264,149.084
C04304=1232.599,-115.302,-35.450,179.430,5.264,149.085
C04305=1232.605,-115.552,-35.440,179.428,5.264,149.085
C04306=1232.609,-115.802,-35.430,179.425,5.264,149.086
C04307=1232.615,-116.051,-35.420,179.423,5.264,149.087
C04308=1232.621,-116.301,-35.411,179.421,5.264,149.087
C04309=1232.626,-116.552,-35.400,179.418,5.264,149.088
C04310=1232.631,-116.801,-35.390,179.417,5.264,149.089
C04311=1232.636,-117.050,-35.380,179.414,5.263,149.089
C04312=1232.641,-117.301,-35.370,179.412,5.264,149.090
C04313=1232.646,-117.550,-35.360,179.409,5.263,149.091
C04314=1232.652,-117.799,-35.350,179.407,5.264,149.092
C04315=1232.657,-118.049,-35.340,179.405,5.263,149.092
C04316=1232.663,-118.300,-35.330,179.402,5.264,149.093
C04317=1232.667,-118.549,-35.320,179.400,5.263,149.094
C04318=1232.673,-118.799,-35.310,179.398,5.264,149.094
C04319=1232.678,-119.049,-35.299,179.396,5.264,149.095
C04320=1232.683,-119.298,-35.290,179.393,5.263,149.096
C04321=1232.688,-119.548,-35.279,179.391,5.264,149.096
C04322=1232.694,-119.798,-35.270,179.389,5.263,149.097
C04323=1232.699,-120.048,-35.260,179.387,5.264,149.098
C04324=1232.704,-120.297,-35.250,179.384,5.263,149.098
C04325=1232.709,-120.546,-35.240,179.382,5.263,149.099
C04326=1232.715,-120.796,-35.230,179.379,5.263,149.100
C04327=1232.720,-121.047,-35.220,179.377,5.263,149.101
C04328=1232.725,-121.296,-35.210,179.374,5.263,149.101
C04329=1232.730,-121.546,-35.200,179.373,5.263,149.102
C04330=1232.736,-121.795,-35.190,179.371,5.263,149.103
C04331=1232.741,-122.046,-35.181,179.368,5.263,149.103
C04332=1232.746,-122.295,-35.171,179.366,5.263,149.104
C04333=1232.751,-122.544,-35.161,179.363,5.263,149.105
C04334=1232.757,-122.794,-35.151,179.361,5.263,149.105
C04335=1232.762,-123.045,-35.141,179.358,5.263,149.106
C04336=1232.767,-123.294,-35.131,179.356,5.263,149.107
C04337=1232.772,-123.544,-35.121,179.354,5.263,149.108
C04338=1232.778,-123.794,-35.112,179.352,5.263,149.108
C04339=1232.783,-124.044,-35.102,179.350,5.263,149.109
C04340=1232.788,-124.293,-35.091,179.347,5.263,149.109
C04341=1232.793,-124.543,-35.082,179.345,5.263,149.110
C04342=1232.799,-124.793,-35.072,179.342,5.263,149.111
C04343=1232.804,-125.042,-35.063,179.340,5.263,149.112
C04344=1232.809,-125.293,-35.053,179.338,5.263,149.112
C04345=1232.814,-125.542,-35.043,179.336,5.263,149.113
C04346=1232.820,-125.792,-35.033,179.334,5.263,149.114
C04347=1232.825,-126.041,-35.024,179.331,5.263,149.114
C04348=1232.403,-126.052,-35.059,179.327,5.266,149.116
C04349=1232.398,-125.802,-35.069,179.329,5.266,149.116
C04350=1232.393,-125.552,-35.078,179.332,5.266,149.115
C04351=1232.387,-125.303,-35.088,179.334,5.266,149.114
C04352=1232.382,-125.054,-35.098,179.336,5.266,149.114
C04353=1232.377,-124.803,-35.108,179.338,5.266,149.113
C04354=1232.372,-124.554,-35.118,179.341,5.267,149.112
C04355=1232.366,-124.304,-35.128,179.343,5.266,149.112
C04356=1232.361,-124.054,-35.137,179.345,5.267,149.111
C04357=1232.356,-123.805,-35.147,179.348,5.266,149.110
C04358=1232.351,-123.554,-35.157,179.350,5.266,149.109
C04359=1232.346,-123.305,-35.166,179.352,5.266,149.109
C04360=1232.340,-123.055,-35.177,179.354,5.266,149.108
C04361=1232.335,-122.806,-35.186,179.357,5.267,149.108
C04362=1232.330,-122.555,-35.196,179.359,5.266,149.107
C04363=1232.324,-122.305,-35.206,179.361,5.267,149.106
C04364=1232.319,-122.056,-35.216,179.363,5.266,149.105
C04365=1232.314,-121.807,-35.226,179.366,5.267,149.105
C04366=1232.309,-121.556,-35.235,179.368,5.267,149.104
C04367=1232.304,-121.307,-35.246,179.370,5.266,149.103
C04368=1232.298,-121.057,-35.256,179.373,5.267,149.103
C04369=1232.293,-120.808,-35.265,179.375,5.267,149.102
C04370=1232.288,-120.557,-35.275,179.377,5.267,149.101
C04371=1232.282,-120.307,-35.285,179.379,5.267,149.101
C04372=1232.277,-120.058,-35.295,179.382,5.267,149.100
C04373=1232.272,-119.809,-35.305,179.384,5.267,149.099
C04374=1232.267,-119.559,-35.315,179.387,5.267,149.098
C04375=1232.262,-119.308,-35.325,179.389,5.267,149.098
C04376=1232.256,-119.059,-35.335,179.391,5.266,149.097
C04377=1232.251,-118.810,-35.345,179.394,5.267,149.096
C04378=1232.246,-118.559,-35.355,179.395,5.267,149.096
C04379=1232.240,-118.310,-35.365,179.398,5.267,149.095
C04380=1232.236,-118.061,-35.375,179.400,5.267,149.094
C04381=1232.230,-117.810,-35.385,179.403,5.267,149.094
C04382=1232.225,-117.560,-35.395,179.405,5.267,149.093
C04383=1232.219,-117.311,-35.405,179.408,5.267,149.092
C04384=1232.214,-117.061,-35.415,179.410,5.267,149.092
C04385=1232.209,-116.811,-35.425,179.412,5.267,149.091
C04386=1232.204,-116.562,-35.436,179.414,5.267,149.090
C04387=1232.199,-116.312,-35.445,179.417,5.267,149.089
C04388=1232.194,-116.062,-35.456,179.419,5.267,149.089
C04389=1232.188,-115.812,-35.465,179.421,5.267,149.088
C04390=1232.182,-115.563,-35.475,179.423,5.268,149.087
C04391=1232.178,-115.313,-35.485,179.426,5.267,149.087
C04392=1232.172,-115.063,-35.496,179.428,5.268,149.086
C04393=1232.167,-114.813,-35.506,179.430,5.267,149.085
C04394=1232.162,-114.563,-35.516,179.433,5.268,149.085
C04395=1232.157,-114.314,-35.526,179.435,5.267,149.084
C04396=1232.151,-114.064,-35.536,179.437,5.267,149.083
C04397=1232.146,-113.814,-35.547,179.440,5.267,149.082
C04398=1232.141,-113.565,-35.557,179.442,5.267,149.082
C04399=1232.136,-113.315,-35.567,179.444,5.268,149.081
C04400=1232.131,-113.065,-35.577,179.446,5.267,149.081
C04401=1232.125,-112.816,-35.587,179.449,5.268,149.080
C04402=1232.120,-112.566,-35.598,179.451,5.267,149.079
C04403=1232.115,-112.316,-35.608,179.454,5.268,149.078
C04404=1232.110,-112.067,-35.618,179.456,5.268,149.078
C04405=1232.104,-111.817,-35.628,179.459,5.268,149.077
C04406=1232.099,-111.567,-35.639,179.461,5.268,149.076
C04407=1232.094,-111.317,-35.649,179.463,5.267,149.076
C04408=1232.089,-111.067,-35.659,179.465,5.268,149.075
C04409=1232.084,-110.818,-35.669,179.467,5.267,149.074
C04410=1232.078,-110.568,-35.679,179.470,5.268,149.073
C04411=1232.073,-110.318,-35.690,179.472,5.268,149.073
C04412=1232.068,-110.068,-35.700,179.474,5.268,149.072
C04413=1232.062,-109.819,-35.710,179.477,5.268,149.071
C04414=1232.057,-109.569,-35.721,179.479,5.268,149.071
C04415=1232.052,-109.319,-35.730,179.481,5.268,149.070
C04416=1232.047,-109.069,-35.741,179.484,5.268,149.069
C04417=1232.042,-108.820,-35.751,179.486,5.268,149.069
C04418=1232.036,-108.570,-35.761,179.489,5.268,149.068
C04419=1232.031,-108.321,-35.773,179.491,5.268,149.067
C04420=1232.026,-108.071,-35.783,179.493,5.268,149.066
C04421=1232.021,-107.821,-35.793,179.496,5.268,149.066
C04422=1232.015,-107.571,-35.804,179.498,5.268,149.065
C04423=1232.011,-107.321,-35.814,179.500,5.268,149.064
C04424=1232.005,-107.072,-35.824,179.502,5.268,149.064
C04425=1232.000,-106.822,-35.834,179.505,5.269,149.063
C04426=1231.995,-106.572,-35.845,179.507,5.268,149.062
C04427=1231.989,-106.323,-35.856,179.509,5.269,149.062
C04428=1231.984,-106.073,-35.866,179.512,5.268,149.061
C04429=1231.979,-105.823,-35.876,179.514,5.269,149.060
C04430=1231.974,-105.573,-35.887,179.516,5.268,149.060
C04431=1231.968,-105.323,-35.897,179.519,5.269,149.059
C04432=1231.963,-105.074,-35.908,179.521,5.269,149.058
C04433=1231.958,-104.824,-35.919,179.523,5.268,149.057
C04434=1231.953,-104.574,-35.929,179.526,5.269,149.057
C04435=1231.947,-104.324,-35.939,179.528,5.268,149.056
C04436=1231.942,-104.075,-35.949,179.531,5.269,149.055
C04437=1231.938,-103.826,-35.960,179.533,5.268,149.055
C04438=1231.932,-103.576,-35.971,179.535,5.269,149.054
C04439=1231.927,-103.326,-35.981,179.537,5.268,149.053
C04440=1231.922,-103.076,-35.991,179.540,5.269,149.053
C04441=1231.917,-102.827,-36.003,179.542,5.269,149.052
C04442=1231.911,-102.577,-36.013,179.544,5.269,149.051
C04443=1231.906,-102.327,-36.023,179.546,5.269,149.050
C04444=1231.901,-102.077,-36.034,179.549,5.269,149.050
C04445=1231.896,-101.828,-36.045,179.551,5.269,149.049
C04446=1231.890,-101.578,-36.055,179.554,5.269,149.048
C04447=1231.885,-101.328,-36.066,179.556,5.269,149.048
C04448=1231.880,-101.079,-36.077,179.558,5.269,149.047
C04449=1231.874,-100.807,-36.088,179.561,5.269,149.046
C04450=1231.869,-100.537,-36.100,179.563,5.270,149.045
C04451=1231.863,-100.266,-36.111,179.566,5.269,149.045
C04452=1231.857,-99.995,-36.123,179.569,5.269,149.044
C04453=1231.852,-99.745,-36.134,179.571,5.269,149.043
C04454=1231.847,-99.495,-36.144,179.574,5.269,149.042
C04455=1231.842,-99.245,-36.155,179.576,5.269,149.042
C04456=1231.836,-98.996,-36.166,179.578,5.269,149.041
C04457=1231.831,-98.746,-36.176,179.580,5.269,149.040
C04458=1231.826,-98.497,-36.187,179.583,5.270,149.040
C04459=1231.821,-98.246,-36.198,179.585,5.269,149.039
C04460=1231.815,-97.997,-36.208,179.588,5.270,149.038
C04461=1231.811,-97.747,-36.219,179.589,5.270,149.038
C04462=1231.806,-97.497,-36.230,179.592,5.270,149.037
C04463=1231.800,-97.248,-36.241,179.594,5.270,149.036
C04464=1231.795,-96.998,-36.251,179.597,5.270,149.036
C04465=1231.790,-96.748,-36.261,179.599,5.270,149.035
C04466=1231.784,-96.498,-36.273,179.602,5.270,149.034
C04467=1231.779,-96.249,-36.283,179.604,5.270,149.033
C04468=1231.774,-95.999,-36.295,179.606,5.270,149.033
C04469=1231.769,-95.749,-36.305,179.609,5.270,149.032
C04470=1231.764,-95.500,-36.316,179.611,5.270,149.031
C04471=1231.759,-95.250,-36.327,179.613,5.270,149.031
C04472=1231.753,-95.001,-36.338,179.615,5.270,149.030
C04473=1231.748,-94.751,-36.348,179.618,5.270,149.029
C04474=1231.742,-94.501,-36.359,179.620,5.270,149.028
C04475=1231.737,-94.251,-36.370,179.623,5.270,149.028
C04476=1231.732,-94.001,-36.381,179.625,5.270,149.027
C04477=1231.727,-93.752,-36.392,179.628,5.270,149.026
C04478=1231.722,-93.502,-36.402,179.630,5.270,149.026
C04479=1231.717,-93.253,-36.413,179.632,5.270,149.025
C04480=1231.711,-93.003,-36.425,179.634,5.270,149.024
C04481=1231.706,-92.753,-36.436,179.637,5.271,149.023
C04482=1231.701,-92.504,-36.447,179.639,5.270,149.023
C04483=1231.696,-92.253,-36.457,179.642,5.271,149.022
C04484=1231.691,-92.004,-36.469,179.644,5.270,149.021
C04485=1231.685,-91.754,-36.479,179.647,5.271,149.021
C04486=1231.680,-91.504,-36.491,179.649,5.270,149.020
C04487=1231.675,-91.255,-36.501,179.651,5.271,149.019
C04488=1231.670,-91.005,-36.512,179.653,5.270,149.018
C04489=1231.665,-90.755,-36.523,179.656,5.271,149.018
C04490=1231.659,-90.506,-36.534,179.658,5.271,149.017
C04491=1231.654,-90.256,-36.546,179.661,5.271,149.016
C04492=1231.649,-90.006,-36.556,179.663,5.271,149.016
C04493=1231.644,-89.757,-36.567,179.665,5.272,149.015
C04494=1231.638,-89.506,-36.578,179.667,5.271,149.014
C04495=1231.634,-89.257,-36.590,179.669,5.271,149.014
C04496=1231.628,-89.008,-36.601,179.672,5.271,149.013
C04497=1231.623,-88.758,-36.611,179.674,5.271,149.012
C04498=1231.618,-88.508,-36.623,179.677,5.271,149.012
C04499=1231.613,-88.259,-36.634,179.679,5.271,149.011
C04500=1231.608,-88.008,-36.644,179.682,5.271,149.010
C04501=1231.603,-87.759,-36.656,179.684,5.271,149.009
C04502=1231.597,-87.510,-36.667,179.686,5.272,149.009
C04503=1231.592,-87.259,-36.678,179.688,5.271,149.008
C04504=1231.587,-87.010,-36.689,179.691,5.272,149.007
C04505=1231.583,-86.760,-36.700,179.693,5.271,149.007
C04506=1231.576,-86.510,-36.711,179.696,5.272,149.006
C04507=1231.572,-86.261,-36.723,179.698,5.271,149.005
C04508=1231.567,-86.011,-36.734,179.701,5.272,149.004
C04509=1231.561,-85.762,-36.745,179.703,5.272,149.004
C04510=1231.556,-85.512,-36.756,179.705,5.272,149.003
C04511=1231.551,-85.262,-36.767,179.708,5.272,149.002
C04512=1231.546,-85.012,-36.779,179.710,5.272,149.002
C04513=1231.540,-84.762,-36.789,179.712,5.272,149.001
C04514=1231.535,-84.513,-36.801,179.715,5.272,149.000
C04515=1231.530,-84.263,-36.812,179.717,5.272,148.999
C04516=1231.525,-84.014,-36.823,179.720,5.272,148.999
C04517=1231.520,-83.764,-36.835,179.722,5.272,148.998
C04518=1231.514,-83.514,-36.846,179.724,5.272,148.997
C04519=1231.510,-83.264,-36.857,179.727,5.272,148.997
C04520=1231.504,-83.015,-36.868,179.729,5.273,148.996
C04521=1231.499,-82.765,-36.880,179.731,5.272,148.995
C04522=1231.494,-82.516,-36.891,179.734,5.273,148.994
C04523=1231.488,-82.265,-36.902,179.736,5.272,148.994
C04524=1231.484,-82.015,-36.914,179.739,5.273,148.993
C04525=1231.478,-81.767,-36.925,179.741,5.272,148.992
C04526=1231.473,-81.517,-36.937,179.744,5.273,148.992
C04527=1231.468,-81.267,-36.948,179.746,5.273,148.991
C04528=1231.463,-81.017,-36.960,179.748,5.273,148.990
C04529=1231.457,-80.767,-36.970,179.750,5.273,148.990
C04530=1231.453,-80.518,-36.981,179.753,5.273,148.989
C04531=1231.447,-80.268,-36.993,179.755,5.273,148.988
C04532=1231.443,-80.018,-37.004,179.758,5.273,148.987
C04533=1231.437,-79.768,-37.016,179.760,5.273,148.987
C04534=1231.432,-79.519,-37.027,179.763,5.273,148.986
C04535=1231.426,-79.270,-37.039,179.765,5.273,148.985
C04536=1231.422,-79.020,-37.050,179.767,5.273,148.985
C04537=1231.417,-78.770,-37.061,179.769,5.273,148.984
C04538=1231.411,-78.520,-37.073,179.772,5.274,148.983
C04539=1231.406,-78.271,-37.084,179.774,5.273,148.982
C04540=1231.401,-78.021,-37.096,179.777,5.274,148.982
C04541=1231.396,-77.771,-37.107,179.779,5.273,148.981
C04542=1231.390,-77.521,-37.119,179.782,5.274,148.980
C04543=1231.386,-77.272,-37.130,179.784,5.273,148.980
C04544=1231.380,-77.022,-37.142,179.786,5.274,148.979
C04545=1231.375,-76.773,-37.153,179.788,5.274,148.978
C04546=1231.370,-76.523,-37.165,179.791,5.274,148.977
C04547=1231.365,-76.273,-37.176,179.793,5.274,148.977
C04548=1231.359,-76.023,-37.188,179.796,5.274,148.976
C04549=1231.355,-75.774,-37.199,179.799,5.275,148.975
C04550=1231.349,-75.524,-37.211,179.801,5.274,148.975
C04551=1231.344,-75.275,-37.222,179.803,5.275,148.974
C04552=1231.339,-75.025,-37.234,179.805,5.274,148.973
C04553=1231.333,-74.755,-37.247,179.808,5.275,148.972
C04554=1231.327,-74.484,-37.259,179.811,5.274,148.972
C04555=1231.322,-74.214,-37.272,179.813,5.275,148.971
C04556=1231.316,-73.944,-37.285,179.816,5.275,148.970
C04557=1231.312,-73.694,-37.296,179.818,5.275,148.969
C04558=1231.306,-73.445,-37.308,179.821,5.275,148.969
C04559=1231.300,-73.195,-37.319,179.823,5.275,148.968
C04560=1231.296,-72.945,-37.331,179.826,5.275,148.967
C04561=1231.290,-72.695,-37.343,179.828,5.275,148.967
C04562=1231.285,-72.446,-37.354,179.830,5.275,148.966
C04563=1231.280,-72.196,-37.366,179.832,5.275,148.965
C04564=1231.275,-71.946,-37.377,179.835,5.276,148.964
C04565=1231.270,-71.696,-37.389,179.837,5.275,148.964
C04566=1231.264,-71.447,-37.400,179.840,5.276,148.963
C04567=1231.259,-71.197,-37.412,179.842,5.275,148.962
C04568=1231.254,-70.948,-37.424,179.845,5.276,148.962
C04569=1231.249,-70.698,-37.436,179.847,5.275,148.961
C04570=1231.244,-70.448,-37.448,179.849,5.276,148.960
C04571=1231.239,-70.198,-37.459,179.851,5.276,148.960
C04572=1231.234,-69.949,-37.471,179.854,5.276,148.959
C04573=1231.228,-69.699,-37.483,179.856,5.276,148.958
C04574=1231.223,-69.449,-37.495,179.859,5.276,148.957
C04575=1231.219,-69.200,-37.506,179.862,5.277,148.957
C04576=1231.213,-68.950,-37.518,179.864,5.276,148.956
C04577=1231.208,-68.700,-37.530,179.866,5.277,148.955
C04578=1231.203,-68.450,-37.542,179.868,5.276,148.955
C04579=1231.197,-68.201,-37.553,179.871,5.277,148.954
C04580=1231.192,-67.952,-37.566,179.873,5.277,148.953
C04581=1231.187,-67.702,-37.577,179.876,5.277,148.952
C04582=1231.182,-67.452,-37.589,179.878,5.276,148.952
C04583=1231.176,-67.202,-37.601,179.881,5.277,148.951
C04584=1231.172,-66.953,-37.613,179.883,5.276,148.950
C04585=1231.167,-66.703,-37.625,179.886,5.277,148.949
C04586=1231.161,-66.453,-37.636,179.888,5.277,148.949
C04587=1231.156,-66.203,-37.648,179.891,5.277,148.948
C04588=1231.151,-65.954,-37.660,179.893,5.277,148.947
C04589=1231.146,-65.705,-37.672,179.895,5.277,148.947
C04590=1231.140,-65.455,-37.684,179.897,5.277,148.946
C04591=1231.136,-65.206,-37.696,179.900,5.277,148.945
C04592=1231.131,-64.956,-37.708,179.903,5.278,148.944
C04593=1231.125,-64.706,-37.720,179.905,5.277,148.944
C04594=1231.120,-64.456,-37.732,179.908,5.278,148.943
C04595=1231.115,-64.207,-37.744,179.910,5.278,148.942
C04596=1231.110,-63.957,-37.756,179.912,5.278,148.942
C04597=1231.104,-63.707,-37.768,179.914,5.278,148.941
C04598=1231.099,-63.458,-37.780,179.917,5.278,148.940
C04599=1231.095,-63.208,-37.791,179.919,5.278,148.939
C04600=1231.089,-62.958,-37.803,179.922,5.278,148.939
C04601=1231.084,-62.709,-37.816,179.924,5.278,148.938
C04602=1231.079,-62.459,-37.828,179.927,5.278,148.937
C04603=1231.074,-62.209,-37.840,179.929,5.278,148.937
C04604=1231.069,-61.960,-37.852,179.931,5.279,148.936
C04605=1231.063,-61.710,-37.864,179.934,5.279,148.935
C04606=1231.058,-61.461,-37.876,179.936,5.279,148.935
C04607=1231.053,-61.211,-37.888,179.939,5.279,148.934
C04608=1231.048,-60.961,-37.901,179.941,5.279,148.933
C04609=1231.043,-60.712,-37.912,179.944,5.279,148.932
C04610=1231.038,-60.462,-37.924,179.946,5.279,148.932
C04611=1231.033,-60.212,-37.937,179.948,5.280,148.931
C04612=1231.028,-59.962,-37.949,179.950,5.279,148.930
C04613=1231.023,-59.712,-37.961,179.953,5.280,148.930
C04614=1231.017,-59.463,-37.973,179.955,5.279,148.929
C04615=1231.013,-59.214,-37.985,179.958,5.280,148.928
C04616=1231.007,-58.964,-37.997,179.960,5.280,148.927
C04617=1231.002,-58.714,-38.010,179.963,5.280,148.927
C04618=1230.997,-58.464,-38.022,179.965,5.280,148.926
C04619=1230.992,-58.215,-38.034,179.967,5.280,148.925
C04620=1230.986,-57.965,-38.046,179.970,5.281,148.925
C04621=1230.981,-57.716,-38.059,179.973,5.280,148.924
C04622=1230.976,-57.466,-38.071,179.975,5.280,148.923
C04623=1230.972,-57.216,-38.083,179.977,5.280,148.922
C04624=1230.966,-56.966,-38.095,179.980,5.281,148.922
C04625=1230.961,-56.717,-38.107,179.983,5.281,148.921
C04626=1230.956,-56.467,-38.119,179.985,5.281,148.920
C04627=1230.951,-56.218,-38.132,179.987,5.281,148.920
C04628=1230.945,-55.968,-38.144,179.989,5.281,148.919
C04629=1230.940,-55.718,-38.156,179.992,5.281,148.918
C04630=1230.935,-55.469,-38.169,179.994,5.281,148.917
C04631=1230.930,-55.219,-38.181,179.997,5.281,148.917
C04632=1230.925,-54.969,-38.194,179.999,5.281,148.916
C04633=1230.920,-54.719,-38.206,-179.998,5.282,148.915
C04634=1230.915,-54.470,-38.218,-179.996,5.282,148.915
C04635=1230.910,-54.221,-38.230,-179.994,5.282,148.914
C04636=1230.905,-53.971,-38.242,-179.991,5.282,148.913
C04637=1230.900,-53.722,-38.255,-179.989,5.282,148.912
C04638=1230.894,-53.472,-38.267,-179.986,5.282,148.912
C04639=1230.890,-53.222,-38.280,-179.984,5.282,148.911
C04640=1230.885,-52.972,-38.292,-179.981,5.283,148.910
C04641=1230.879,-52.722,-38.304,-179.979,5.282,148.910
C04642=1230.874,-52.473,-38.317,-179.977,5.283,148.909
C04643=1230.869,-52.224,-38.329,-179.974,5.283,148.908
C04644=1230.863,-51.974,-38.341,-179.972,5.283,148.908
C04645=1230.859,-51.724,-38.354,-179.969,5.283,148.907
C04646=1230.854,-51.474,-38.367,-179.967,5.283,148.906
C04647=1230.848,-51.225,-38.379,-179.965,5.284,148.905
C04648=1230.843,-50.975,-38.391,-179.962,5.283,148.905
C04649=1230.838,-50.726,-38.404,-179.960,5.284,148.904
C04650=1230.833,-50.476,-38.416,-179.957,5.284,148.903
C04651=1230.828,-50.226,-38.429,-179.955,5.284,148.903
C04652=1230.823,-49.977,-38.441,-179.952,5.284,148.902
C04653=1230.818,-49.727,-38.454,-179.950,5.284,148.901
C04654=1230.813,-49.477,-38.466,-179.947,5.284,148.900
C04655=1230.807,-49.228,-38.478,-179.945,5.284,148.900
C04656=1230.802,-48.978,-38.492,-179.942,5.284,148.899
C04657=1230.797,-48.709,-38.505,-179.940,5.285,148.898
C04658=1230.791,-48.438,-38.518,-179.938,5.284,148.897
C04659=1230.785,-48.168,-38.533,-179.934,5.285,148.897
C04660=1230.780,-47.899,-38.546,-179.932,5.285,148.896
C04661=1230.775,-47.649,-38.559,-179.930,5.285,148.895
C04662=1230.770,-47.400,-38.571,-179.927,5.285,148.894
C04663=1230.765,-47.150,-38.583,-179.924,5.286,148.894
C04664=1230.760,-46.901,-38.596,-179.922,5.285,148.893
C04665=1230.755,-46.651,-38.609,-179.920,5.286,148.892
C04666=1230.749,-46.401,-38.622,-179.918,5.286,148.892
C04667=1230.744,-46.152,-38.635,-179.915,5.286,148.891
C04668=1230.739,-45.902,-38.647,-179.913,5.286,148.890
C04669=1230.734,-45.652,-38.659,-179.910,5.286,148.890
C04670=1230.729,-45.402,-38.672,-179.907,5.287,148.889
C04671=1230.724,-45.153,-38.685,-179.905,5.286,148.888
C04672=1230.719,-44.904,-38.697,-179.903,5.287,148.887
C04673=1230.714,-44.653,-38.711,-179.901,5.286,148.887
C04674=1230.708,-44.404,-38.724,-179.898,5.287,148.886
C04675=1230.703,-44.155,-38.736,-179.896,5.287,148.885
C04676=1230.698,-43.905,-38.748,-179.893,5.287,148.885
C04677=1230.693,-43.655,-38.761,-179.891,5.288,148.884
C04678=1230.688,-43.406,-38.774,-179.888,5.287,148.883
C04679=1230.682,-43.156,-38.787,-179.886,5.288,148.883
C04680=1230.677,-42.907,-38.799,-179.883,5.287,148.882
C04681=1230.673,-42.657,-38.812,-179.881,5.288,148.881
C04682=1230.668,-42.407,-38.825,-179.878,5.288,148.880
C04683=1230.663,-42.158,-38.838,-179.876,5.288,148.879
C04684=1230.657,-41.908,-38.851,-179.873,5.288,148.879
C04685=1230.652,-41.658,-38.864,-179.871,5.288,148.878
C04686=1230.647,-41.409,-38.876,-179.868,5.288,148.877
C04687=1230.642,-41.159,-38.889,-179.866,5.289,148.877
C04688=1230.637,-40.910,-38.902,-179.864,5.289,148.876
C04689=1230.631,-40.660,-38.915,-179.861,5.289,148.875
C04690=1230.627,-40.410,-38.928,-179.859,5.289,148.875
C04691=1230.622,-40.161,-38.941,-179.856,5.289,148.874
C04692=1230.617,-39.911,-38.953,-179.854,5.290,148.873
C04693=1230.611,-39.661,-38.967,-179.851,5.289,148.872
C04694=1230.606,-39.412,-38.979,-179.849,5.290,148.872
C04695=1230.601,-39.162,-38.992,-179.847,5.290,148.871
C04696=1230.597,-38.912,-39.005,-179.844,5.290,148.870
C04697=1230.591,-38.663,-39.018,-179.841,5.291,148.870
C04698=1230.586,-38.413,-39.031,-179.839,5.290,148.869
C04699=1230.581,-38.163,-39.044,-179.837,5.291,148.868
C04700=1230.575,-37.914,-39.057,-179.835,5.290,148.868
C04701=1230.570,-37.665,-39.070,-179.832,5.291,148.867
C04702=1230.566,-37.415,-39.083,-179.829,5.291,148.866
C04703=1230.560,-37.165,-39.096,-179.827,5.291,148.865
C04704=1230.555,-36.916,-39.109,-179.824,5.292,148.865
C04705=1230.550,-36.666,-39.122,-179.822,5.291,148.864
C04706=1230.545,-36.417,-39.135,-179.819,5.291,148.863
C04707=1230.540,-36.166,-39.148,-179.817,5.292,148.862
C04708=1230.535,-35.917,-39.161,-179.814,5.292,148.862
C04709=1230.530,-35.668,-39.173,-179.812,5.292,148.861
C04710=1230.525,-35.418,-39.188,-179.810,5.292,148.860
C04711=1230.520,-35.169,-39.200,-179.807,5.292,148.860
C04712=1230.515,-34.919,-39.214,-179.804,5.293,148.859
C04713=1230.509,-34.669,-39.226,-179.802,5.293,148.858
C04714=1230.504,-34.420,-39.239,-179.800,5.293,148.858
C04715=1230.499,-34.170,-39.253,-179.798,5.293,148.857
C04716=1230.494,-33.921,-39.266,-179.795,5.293,148.856
C04717=1230.490,-33.671,-39.279,-179.792,5.294,148.855
C04718=1230.484,-33.421,-39.292,-179.790,5.293,148.855
C04719=1230.479,-33.172,-39.305,-179.788,5.294,148.854
C04720=1230.473,-32.922,-39.318,-179.785,5.294,148.853
C04721=1230.469,-32.673,-39.331,-179.783,5.294,148.853
C04722=1230.464,-32.423,-39.344,-179.780,5.295,148.852
C04723=1230.458,-32.173,-39.358,-179.778,5.294,148.851
C04724=1230.454,-31.923,-39.371,-179.775,5.295,148.851
C04725=1230.448,-31.674,-39.385,-179.773,5.295,148.850
C04726=1230.443,-31.425,-39.397,-179.771,5.295,148.849
C04727=1230.438,-31.175,-39.411,-179.768,5.295,148.848
C04728=1230.433,-30.926,-39.424,-179.766,5.295,148.848
C04729=1230.428,-30.676,-39.437,-179.763,5.296,148.847
C04730=1230.423,-30.426,-39.450,-179.761,5.296,148.846
C04731=1230.418,-30.176,-39.463,-179.758,5.296,148.846
C04732=1230.412,-29.927,-39.477,-179.755,5.296,148.845
C04733=1230.408,-29.677,-39.490,-179.753,5.296,148.844
C04734=1230.402,-29.428,-39.503,-179.751,5.296,148.843
C04735=1230.398,-29.178,-39.517,-179.748,5.297,148.843
C04736=1230.392,-28.928,-39.530,-179.746,5.296,148.842
C04737=1230.387,-28.678,-39.543,-179.743,5.297,148.841
C04738=1230.382,-28.429,-39.557,-179.740,5.297,148.841
C04739=1230.377,-28.179,-39.570,-179.738,5.297,148.840
C04740=1230.372,-27.930,-39.584,-179.736,5.298,148.839
C04741=1230.367,-27.680,-39.597,-179.733,5.298,148.838
C04742=1230.361,-27.431,-39.610,-179.731,5.298,148.838
C04743=1230.357,-27.181,-39.624,-179.728,5.298,148.837
C04744=1230.351,-26.932,-39.637,-179.726,5.298,148.836
C04745=1230.347,-26.682,-39.651,-179.724,5.298,148.836
C04746=1230.341,-26.433,-39.664,-179.721,5.299,148.835
C04747=1230.337,-26.183,-39.677,-179.719,5.299,148.834
C04748=1230.331,-25.934,-39.691,-179.716,5.299,148.834
C04749=1230.327,-25.684,-39.704,-179.714,5.300,148.833
C04750=1230.321,-25.435,-39.718,-179.711,5.299,148.832
C04751=1230.316,-25.184,-39.731,-179.709,5.300,148.831
C04752=1230.311,-24.936,-39.744,-179.706,5.300,148.831
C04753=1230.306,-24.685,-39.758,-179.704,5.300,148.830
C04754=1230.302,-24.436,-39.772,-179.701,5.301,148.829
C04755=1230.296,-24.186,-39.785,-179.699,5.300,148.829
C04756=1230.292,-23.937,-39.799,-179.697,5.301,148.828
C04757=1230.286,-23.687,-39.812,-179.694,5.301,148.827
C04758=1230.281,-23.438,-39.826,-179.692,5.301,148.827
C04759=1230.276,-23.188,-39.839,-179.689,5.301,148.826
C04760=1230.271,-22.939,-39.853,-179.686,5.302,148.825
C04761=1230.265,-22.668,-39.867,-179.684,5.301,148.824
C04762=1230.260,-22.400,-39.881,-179.681,5.302,148.824
C04763=1230.254,-22.131,-39.896,-179.679,5.302,148.823
C04764=1230.249,-21.861,-39.911,-179.676,5.302,148.822
C04765=1230.244,-21.612,-39.925,-179.673,5.302,148.821
C04766=1230.239,-21.362,-39.938,-179.671,5.303,148.821
C04767=1230.234,-21.113,-39.952,-179.668,5.303,148.820
C04768=1230.229,-20.863,-39.965,-179.666,5.303,148.819
C04769=1230.224,-20.613,-39.979,-179.663,5.303,148.818
C04770=1230.218,-20.364,-39.992,-179.661,5.304,148.818
C04771=1230.214,-20.114,-40.006,-179.659,5.304,148.817
C04772=1230.209,-19.865,-40.020,-179.656,5.304,148.816
C04773=1230.203,-19.615,-40.034,-179.653,5.305,148.816
C04774=1230.198,-19.365,-40.048,-179.651,5.304,148.815
C04775=1230.194,-19.116,-40.062,-179.649,5.305,148.814
C04776=1230.188,-18.866,-40.075,-179.646,5.305,148.814
C04777=1230.183,-18.617,-40.089,-179.644,5.305,148.813
C04778=1230.178,-18.368,-40.102,-179.641,5.306,148.812
C04779=1230.173,-18.118,-40.116,-179.639,5.306,148.812
C04780=1230.168,-17.868,-40.130,-179.636,5.306,148.811
C04781=1230.163,-17.619,-40.143,-179.634,5.306,148.810
C04782=1230.158,-17.369,-40.157,-179.631,5.307,148.809
C04783=1230.153,-17.119,-40.171,-179.629,5.306,148.809
C04784=1230.147,-16.870,-40.185,-179.626,5.307,148.808
C04785=1230.143,-16.620,-40.198,-179.624,5.307,148.807
C04786=1230.138,-16.370,-40.212,-179.622,5.307,148.807
C04787=1230.132,-16.121,-40.226,-179.619,5.308,148.806
C04788=1230.127,-15.872,-40.241,-179.616,5.308,148.805
C04789=1230.123,-15.622,-40.254,-179.614,5.308,148.805
C04790=1230.117,-15.373,-40.268,-179.612,5.308,148.804
C04791=1230.112,-15.123,-40.282,-179.609,5.309,148.803
C04792=1230.107,-14.873,-40.296,-179.607,5.309,148.803
C04793=1230.101,-14.624,-40.309,-179.604,5.309,148.802
C04794=1230.097,-14.374,-40.323,-179.601,5.309,148.801
C04795=1230.092,-14.125,-40.337,-179.599,5.309,148.800
C04796=1230.087,-13.876,-40.351,-179.596,5.310,148.799
C04797=1230.081,-13.625,-40.365,-179.594,5.310,148.799
C04798=1230.076,-13.375,-40.379,-179.592,5.310,148.798
C04799=1230.071,-13.127,-40.392,-179.589,5.310,148.797
C04800=1230.067,-12.877,-40.407,-179.586,5.311,148.797
C04801=1230.062,-12.627,-40.421,-179.584,5.310,148.796
C04802=1230.057,-12.378,-40.435,-179.582,5.311,148.795
C04803=1230.051,-12.128,-40.448,-179.579,5.311,148.795
C04804=1230.046,-11.878,-40.463,-179.577,5.311,148.794
C04805=1230.042,-11.629,-40.476,-179.574,5.312,148.793
C04806=1230.037,-11.379,-40.491,-179.572,5.312,148.793
C04807=1230.031,-11.130,-40.504,-179.569,5.312,148.792
C04808=1230.026,-10.880,-40.519,-179.567,5.312,148.791
C04809=1230.021,-10.631,-40.533,-179.564,5.313,148.790
C04810=1230.016,-10.382,-40.547,-179.562,5.313,148.790
C04811=1230.011,-10.132,-40.561,-179.559,5.313,148.789
C04812=1230.005,-9.882,-40.575,-179.557,5.314,148.788
C04813=1230.001,-9.632,-40.588,-179.554,5.314,148.788
C04814=1229.996,-9.383,-40.603,-179.552,5.314,148.787
C04815=1229.991,-9.134,-40.617,-179.549,5.314,148.786
C04816=1229.986,-8.884,-40.631,-179.547,5.315,148.786
C04817=1229.981,-8.634,-40.645,-179.545,5.315,148.785
C04818=1229.976,-8.384,-40.659,-179.542,5.315,148.784
C04819=1229.970,-8.135,-40.673,-179.539,5.316,148.784
C04820=1229.965,-7.886,-40.688,-179.537,5.315,148.783
C04821=1229.960,-7.636,-40.702,-179.535,5.316,148.782
C04822=1229.955,-7.386,-40.716,-179.532,5.316,148.781
C04823=1229.950,-7.137,-40.730,-179.530,5.316,148.781
C04824=1229.945,-6.888,-40.744,-179.527,5.317,148.780
C04825=1229.940,-6.638,-40.759,-179.525,5.317,148.779
C04826=1229.936,-6.389,-40.772,-179.522,5.318,148.779
C04827=1229.931,-6.139,-40.787,-179.520,5.317,148.778
C04828=1229.926,-5.889,-40.801,-179.517,5.318,148.777
C04829=1229.920,-5.640,-40.815,-179.514,5.318,148.777
C04830=1229.915,-5.390,-40.829,-179.512,5.318,148.776
C04831=1229.910,-5.141,-40.843,-179.510,5.319,148.775
C04832=1229.905,-4.891,-40.858,-179.507,5.319,148.775
C04833=1229.901,-4.642,-40.873,-179.505,5.319,148.774
C04834=1229.896,-4.392,-40.887,-179.502,5.319,148.773
C04835=1229.890,-4.143,-40.901,-179.500,5.320,148.773
C04836=1229.885,-3.893,-40.915,-179.497,5.321,148.772
C04837=1229.880,-3.644,-40.929,-179.495,5.320,148.771
C04838=1229.875,-3.394,-40.944,-179.492,5.321,148.770
C04839=1229.870,-3.144,-40.959,-179.490,5.321,148.770
C04840=1229.865,-2.894,-40.973,-179.488,5.321,148.769
C04841=1229.859,-2.645,-40.987,-179.485,5.322,148.768
C04842=1229.855,-2.396,-41.002,-179.482,5.322,148.767
C04843=1229.850,-2.146,-41.016,-179.479,5.322,148.767
C04844=1229.845,-1.897,-41.030,-179.477,5.322,148.766
C04845=1229.840,-1.647,-41.045,-179.474,5.322,148.765
C04846=1229.835,-1.397,-41.059,-179.472,5.323,148.765
C04847=1229.830,-1.148,-41.073,-179.470,5.323,148.764
C04848=1229.824,-0.899,-41.088,-179.467,5.323,148.763
C04849=1229.820,-0.650,-41.102,-179.464,5.324,148.763
C04850=1229.815,-0.400,-41.116,-179.462,5.324,148.762
C04851=1229.810,-0.150,-41.131,-179.460,5.324,148.761
C04852=1229.805,0.100,-41.145,-179.457,5.324,148.761
C04853=1229.799,0.349,-41.160,-179.454,5.325,148.760
C04854=1229.794,0.599,-41.175,-179.452,5.325,148.759
C04855=1229.789,0.848,-41.189,-179.450,5.325,148.758
C04856=1229.784,1.098,-41.203,-179.447,5.326,148.758
C04857=1229.780,1.347,-41.218,-179.444,5.326,148.757
C04858=1229.774,1.596,-41.232,-179.442,5.326,148.756
C04859=1229.769,1.846,-41.246,-179.440,5.327,148.756
C04860=1229.764,2.095,-41.262,-179.437,5.327,148.755
C04861=1229.759,2.345,-41.276,-179.434,5.328,148.754
C04862=1229.754,2.595,-41.291,-179.432,5.327,148.754
C04863=1229.749,2.845,-41.305,-179.430,5.328,148.753
C04864=1229.744,3.094,-41.320,-179.427,5.328,148.752
C04865=1229.739,3.362,-41.336,-179.424,5.329,148.752
C04866=1229.733,3.632,-41.351,-179.422,5.329,148.751
C04867=1229.728,3.901,-41.367,-179.419,5.329,148.750
C04868=1229.723,4.170,-41.383,-179.416,5.329,148.749
C04869=1229.718,4.419,-41.398,-179.414,5.330,148.749
C04870=1229.712,4.669,-41.412,-179.411,5.330,148.748
C04871=1229.708,4.919,-41.427,-179.409,5.330,148.747
C04872=1229.703,5.168,-41.442,-179.406,5.331,148.747
C04873=1229.698,5.417,-41.456,-179.404,5.331,148.746
C04874=1229.692,5.667,-41.471,-179.401,5.332,148.745
C04875=1229.688,5.916,-41.486,-179.399,5.331,148.744
C04876=1229.682,6.165,-41.500,-179.396,5.332,148.744
C04877=1229.677,6.415,-41.515,-179.394,5.332,148.743
C04878=1229.672,6.664,-41.529,-179.391,5.333,148.742
C04879=1229.667,6.914,-41.545,-179.389,5.333,148.742
C04880=1229.662,7.163,-41.559,-179.386,5.333,148.741
C04881=1229.657,7.413,-41.573,-179.384,5.334,148.740
C04882=1229.652,7.662,-41.589,-179.381,5.334,148.740
C04883=1229.647,7.912,-41.603,-179.379,5.334,148.739
C04884=1229.642,8.161,-41.618,-179.376,5.335,148.738
C04885=1229.637,8.411,-41.632,-179.374,5.335,148.738
C04886=1229.632,8.661,-41.648,-179.371,5.336,148.737
C04887=1229.627,8.911,-41.663,-179.369,5.335,148.736
C04888=1229.623,9.160,-41.678,-179.366,5.336,148.736
C04889=1229.617,9.410,-41.692,-179.364,5.336,148.735
C04890=1229.612,9.659,-41.707,-179.361,5.337,148.734
C04891=1229.607,9.909,-41.722,-179.359,5.337,148.734
C04892=1229.602,10.158,-41.737,-179.356,5.337,148.733
C04893=1229.597,10.407,-41.752,-179.354,5.338,148.732
C04894=1229.592,10.657,-41.767,-179.351,5.338,148.731
C04895=1229.587,10.906,-41.782,-179.349,5.338,148.731
C04896=1229.582,11.156,-41.796,-179.346,5.339,148.730
C04897=1229.577,11.405,-41.811,-179.343,5.339,148.729
C04898=1229.572,11.655,-41.826,-179.341,5.340,148.729
C04899=1229.567,11.904,-41.841,-179.339,5.340,148.728
C04900=1229.563,12.153,-41.856,-179.337,5.340,148.728
C04901=1229.557,12.403,-41.871,-179.334,5.341,148.727
C04902=1229.552,12.652,-41.886,-179.331,5.341,148.726
C04903=1229.546,12.902,-41.901,-179.329,5.342,148.726
C04904=1229.542,13.152,-41.916,-179.327,5.342,148.725
C04905=1229.538,13.401,-41.931,-179.324,5.342,148.724
C04906=1229.532,13.651,-41.946,-179.321,5.343,148.723
C04907=1229.527,13.900,-41.961,-179.319,5.343,148.723
C04908=1229.522,14.150,-41.977,-179.317,5.343,148.722
C04909=1229.517,14.400,-41.991,-179.314,5.343,148.721
C04910=1229.512,14.649,-42.006,-179.311,5.344,148.721
C04911=1229.507,14.898,-42.022,-179.309,5.345,148.720
C04912=1229.502,15.148,-42.036,-179.307,5.344,148.719
C04913=1229.497,15.397,-42.052,-179.304,5.345,148.719
C04914=1229.492,15.646,-42.067,-179.301,5.345,148.718
C04915=1229.487,15.896,-42.082,-179.299,5.346,148.717
C04916=1229.482,16.146,-42.097,-179.296,5.346,148.717
C04917=1229.477,16.395,-42.112,-179.294,5.346,148.716
C04918=1229.472,16.645,-42.127,-179.291,5.347,148.715
C04919=1229.467,16.895,-42.142,-179.289,5.347,148.715
C04920=1229.462,17.144,-42.157,-179.286,5.348,148.714
C04921=1229.457,17.393,-42.172,-179.284,5.347,148.713
C04922=1229.453,17.643,-42.188,-179.281,5.348,148.713
C04923=1229.448,17.892,-42.203,-179.279,5.349,148.712
C04924=1229.442,18.142,-42.218,-179.276,5.349,148.711
C04925=1229.438,18.391,-42.233,-179.273,5.350,148.710
C04926=1229.432,18.640,-42.249,-179.271,5.349,148.710
C04927=1229.427,18.890,-42.264,-179.269,5.350,148.709
C04928=1229.423,19.140,-42.280,-179.266,5.350,148.708
C04929=1229.417,19.390,-42.294,-179.263,5.351,148.708
C04930=1229.412,19.639,-42.309,-179.261,5.352,148.707
C04931=1229.407,19.888,-42.325,-179.259,5.351,148.706
C04932=1229.402,20.137,-42.340,-179.256,5.352,148.706
C04933=1229.397,20.387,-42.356,-179.253,5.352,148.705
C04934=1229.393,20.636,-42.371,-179.251,5.353,148.704
C04935=1229.387,20.886,-42.386,-179.248,5.353,148.704
C04936=1229.383,21.136,-42.401,-179.246,5.353,148.703
C04937=1229.377,21.385,-42.416,-179.243,5.354,148.702
C04938=1229.372,21.634,-42.432,-179.241,5.354,148.702
C04939=1229.368,21.884,-42.447,-179.238,5.355,148.701
C04940=1229.362,22.134,-42.463,-179.235,5.355,148.700
C04941=1229.358,22.383,-42.478,-179.233,5.355,148.700
C04942=1229.352,22.632,-42.493,-179.231,5.356,148.699
C04943=1229.347,22.881,-42.509,-179.228,5.357,148.698
C04944=1229.343,23.131,-42.524,-179.226,5.357,148.698
C04945=1229.337,23.381,-42.540,-179.223,5.358,148.697
C04946=1229.333,23.630,-42.555,-179.221,5.357,148.696
C04947=1229.327,23.879,-42.571,-179.218,5.358,148.696
C04948=1229.323,24.129,-42.587,-179.216,5.358,148.695
C04949=1229.318,24.378,-42.602,-179.213,5.359,148.694
C04950=1229.313,24.628,-42.617,-179.210,5.360,148.694
C04951=1229.307,24.877,-42.633,-179.208,5.359,148.693
C04952=1229.303,25.127,-42.648,-179.206,5.360,148.692
C04953=1229.298,25.376,-42.664,-179.203,5.360,148.692
C04954=1229.292,25.626,-42.679,-179.200,5.361,148.691
C04955=1229.288,25.875,-42.694,-179.198,5.361,148.690
C04956=1229.283,26.125,-42.710,-179.195,5.362,148.690
C04957=1229.278,26.374,-42.726,-179.193,5.362,148.689
C04958=1229.273,26.623,-42.741,-179.190,5.362,148.688
C04959=1229.268,26.874,-42.757,-179.188,5.363,148.688
C04960=1229.263,27.123,-42.772,-179.185,5.363,148.687
C04961=1229.257,27.372,-42.788,-179.183,5.364,148.686
C04962=1229.253,27.621,-42.803,-179.180,5.364,148.685
C04963=1229.248,27.872,-42.819,-179.178,5.364,148.685
C04964=1229.243,28.121,-42.834,-179.175,5.365,148.684
C04965=1229.238,28.369,-42.850,-179.173,5.365,148.683
C04966=1229.233,28.620,-42.866,-179.170,5.366,148.683
C04967=1229.228,28.869,-42.882,-179.168,5.367,148.682
C04968=1229.223,29.118,-42.897,-179.166,5.367,148.682
C04969=1229.217,29.387,-42.914,-179.163,5.367,148.681
C04970=1229.213,29.656,-42.931,-179.160,5.367,148.680
C04971=1229.207,29.924,-42.948,-179.157,5.368,148.679
C04972=1229.201,30.193,-42.964,-179.155,5.368,148.679
C04973=1229.196,30.442,-42.981,-179.152,5.369,148.678
C04974=1229.192,30.692,-42.997,-179.149,5.370,148.677
C04975=1229.187,30.941,-43.012,-179.147,5.370,148.677
C04976=1229.182,31.191,-43.027,-179.144,5.371,148.676
C04977=1229.177,31.441,-43.043,-179.141,5.371,148.675
C04978=1229.172,31.690,-43.059,-179.139,5.371,148.675
C04979=1229.166,31.939,-43.075,-179.137,5.371,148.674
C04980=1229.162,32.189,-43.090,-179.134,5.372,148.673
C04981=1229.157,32.438,-43.106,-179.131,5.373,148.673
C04982=1229.152,32.687,-43.122,-179.129,5.373,148.672
C04983=1229.147,32.937,-43.138,-179.127,5.374,148.671
C04984=1229.142,33.186,-43.154,-179.124,5.374,148.671
C04985=1229.137,33.437,-43.170,-179.122,5.374,148.670
C04986=1229.132,33.685,-43.186,-179.119,5.375,148.669
C04987=1229.127,33.934,-43.201,-179.117,5.375,148.669
C04988=1229.122,34.185,-43.217,-179.114,5.376,148.668
C04989=1229.117,34.433,-43.233,-179.111,5.377,148.667
C04990=1229.112,34.683,-43.249,-179.109,5.377,148.667
C04991=1229.107,34.933,-43.265,-179.107,5.377,148.666
C04992=1229.102,35.182,-43.281,-179.104,5.377,148.665
C04993=1229.097,35.432,-43.297,-179.101,5.378,148.665
C04994=1229.093,35.681,-43.312,-179.099,5.379,148.664
C04995=1229.088,35.930,-43.329,-179.096,5.379,148.663
C04996=1229.083,36.180,-43.344,-179.093,5.380,148.663
C04997=1229.077,36.429,-43.360,-179.091,5.381,148.662
C04998=1229.073,36.679,-43.377,-179.089,5.380,148.662
C04999=1229.067,36.928,-43.392,-179.086,5.381,148.661
C05000=1229.063,37.177,-43.409,-179.084,5.381,148.660
C05001=1229.058,37.427,-43.425,-179.081,5.382,148.660
C05002=1229.053,37.677,-43.440,-179.079,5.383,148.659
C05003=1229.048,37.926,-43.457,-179.076,5.383,148.658
C05004=1229.043,38.176,-43.473,-179.073,5.384,148.658
C05005=1229.038,38.425,-43.489,-179.071,5.384,148.657
C05006=1229.032,38.674,-43.505,-179.069,5.384,148.656
C05007=1229.028,38.923,-43.521,-179.066,5.385,148.655
C05008=1229.023,39.173,-43.537,-179.063,5.385,148.655
C05009=1229.018,39.422,-43.554,-179.061,5.386,148.654
C05010=1229.013,39.672,-43.569,-179.059,5.387,148.654
C05011=1229.008,39.921,-43.586,-179.056,5.387,148.653
C05012=1229.003,40.171,-43.601,-179.053,5.388,148.652
C05013=1228.998,40.420,-43.618,-179.051,5.388,148.652
C05014=1228.993,40.670,-43.634,-179.049,5.388,148.651
C05015=1228.988,40.919,-43.650,-179.046,5.389,148.650
C05016=1228.983,41.168,-43.666,-179.043,5.389,148.650
C05017=1228.979,41.418,-43.683,-179.041,5.390,148.649
C05018=1228.973,41.667,-43.698,-179.038,5.390,148.648
C05019=1228.969,41.917,-43.715,-179.035,5.391,148.648
C05020=1228.963,42.166,-43.730,-179.033,5.391,148.647
C05021=1228.959,42.416,-43.747,-179.031,5.392,148.647
C05022=1228.954,42.664,-43.763,-179.028,5.392,148.646
C05023=1228.949,42.915,-43.779,-179.026,5.393,148.645
C05024=1228.944,43.163,-43.796,-179.023,5.393,148.644
C05025=1228.939,43.413,-43.812,-179.021,5.394,148.644
C05026=1228.934,43.662,-43.828,-179.018,5.394,148.643
C05027=1228.929,43.912,-43.845,-179.015,5.395,148.642
C05028=1228.923,44.161,-43.861,-179.013,5.395,148.642
C05029=1228.919,44.411,-43.877,-179.010,5.396,148.641
C05030=1228.914,44.660,-43.893,-179.007,5.397,148.640
C05031=1228.909,44.910,-43.910,-179.005,5.397,148.640
C05032=1228.905,45.159,-43.926,-179.003,5.397,148.639
C05033=1228.899,45.409,-43.942,-179.001,5.398,148.639
C05034=1228.895,45.658,-43.959,-178.998,5.398,148.638
C05035=1228.890,45.907,-43.975,-178.995,5.399,148.637
C05036=1228.884,46.157,-43.992,-178.993,5.399,148.637
C05037=1228.879,46.406,-44.008,-178.990,5.400,148.636
C05038=1228.875,46.656,-44.024,-178.987,5.401,148.635
C05039=1228.870,46.905,-44.041,-178.985,5.401,148.635
C05040=1228.865,47.155,-44.057,-178.982,5.402,148.634
C05041=1228.860,47.404,-44.073,-178.979,5.402,148.633
C05042=1228.854,47.653,-44.090,-178.978,5.402,148.633
C05043=1228.850,47.903,-44.107,-178.975,5.403,148.632
C05044=1228.845,48.153,-44.123,-178.973,5.404,148.631
C05045=1228.840,48.401,-44.139,-178.970,5.404,148.631
C05046=1228.836,48.651,-44.156,-178.967,5.405,148.630
C05047=1228.830,48.900,-44.173,-178.965,5.405,148.629
C05048=1228.825,49.150,-44.189,-178.962,5.406,148.629
C05049=1228.821,49.400,-44.205,-178.959,5.406,148.628
C05050=1228.815,49.648,-44.222,-178.957,5.407,148.627
C05051=1228.811,49.898,-44.238,-178.955,5.408,148.627
C05052=1228.805,50.147,-44.255,-178.952,5.408,148.626
C05053=1228.801,50.397,-44.272,-178.949,5.409,148.626
C05054=1228.796,50.646,-44.289,-178.947,5.410,148.625
C05055=1228.791,50.895,-44.304,-178.945,5.409,148.624
C05056=1228.786,51.145,-44.321,-178.942,5.410,148.624
C05057=1228.781,51.395,-44.338,-178.939,5.410,148.623
C05058=1228.776,51.643,-44.354,-178.937,5.411,148.622
C05059=1228.772,51.893,-44.371,-178.935,5.412,148.622
C05060=1228.766,52.143,-44.388,-178.932,5.413,148.621
C05061=1228.761,52.392,-44.405,-178.929,5.413,148.621
C05062=1228.757,52.641,-44.421,-178.927,5.414,148.620
C05063=1228.752,52.891,-44.439,-178.924,5.414,148.619
C05064=1228.746,53.140,-44.454,-178.921,5.415,148.619
C05065=1228.742,53.390,-44.471,-178.919,5.415,148.618
C05066=1228.737,53.639,-44.488,-178.916,5.416,148.617
C05067=1228.731,53.888,-44.504,-178.914,5.417,148.617
C05068=1228.727,54.138,-44.521,-178.911,5.417,148.616
C05069=1228.722,54.387,-44.538,-178.909,5.417,148.615
C05070=1228.717,54.636,-44.555,-178.907,5.418,148.615
C05071=1228.712,54.886,-44.571,-178.904,5.418,148.614
C05072=1228.707,55.136,-44.589,-178.901,5.419,148.613
C05073=1228.702,55.403,-44.606,-178.899,5.419,148.613
C05074=1228.697,55.672,-44.624,-178.896,5.421,148.612
C05075=1228.691,55.940,-44.643,-178.893,5.421,148.611
C05076=1228.686,56.209,-44.661,-178.890,5.422,148.611
C05077=1228.681,56.459,-44.678,-178.888,5.423,148.610
C05078=1228.676,56.707,-44.694,-178.885,5.423,148.609
C05079=1228.672,56.957,-44.711,-178.882,5.424,148.609
C05080=1228.666,57.207,-44.728,-178.880,5.424,148.608
C05081=1228.662,57.456,-44.745,-178.878,5.424,148.608
C05082=1228.656,57.705,-44.762,-178.876,5.425,148.607
C05083=1228.652,57.955,-44.779,-178.873,5.426,148.606
C05084=1228.647,58.204,-44.795,-178.870,5.426,148.606
C05085=1228.642,58.454,-44.813,-178.868,5.427,148.605
C05086=1228.637,58.703,-44.829,-178.865,5.427,148.604
C05087=1228.632,58.952,-44.847,-178.862,5.428,148.604
C05088=1228.627,59.201,-44.863,-178.860,5.429,148.603
C05089=1228.622,59.451,-44.881,-178.858,5.429,148.603
C05090=1228.617,59.700,-44.897,-178.855,5.430,148.602
C05091=1228.612,59.950,-44.914,-178.852,5.431,148.601
C05092=1228.607,60.199,-44.931,-178.850,5.431,148.601
C05093=1228.602,60.449,-44.948,-178.847,5.432,148.600
C05094=1228.598,60.698,-44.966,-178.844,5.432,148.599
C05095=1228.592,60.947,-44.983,-178.842,5.433,148.599
C05096=1228.588,61.196,-44.999,-178.840,5.434,148.598
C05097=1228.583,61.446,-45.016,-178.837,5.434,148.597
C05098=1228.578,61.696,-45.033,-178.834,5.435,148.597
C05099=1228.573,61.944,-45.051,-178.832,5.436,148.596
C05100=1228.568,62.194,-45.067,-178.829,5.436,148.595
C05101=1228.563,62.444,-45.085,-178.827,5.437,148.595
C05102=1228.558,62.693,-45.101,-178.824,5.438,148.594
C05103=1228.553,62.942,-45.119,-178.822,5.438,148.594
C05104=1228.549,63.192,-45.136,-178.819,5.439,148.593
C05105=1228.543,63.441,-45.153,-178.816,5.439,148.592
C05106=1228.539,63.690,-45.170,-178.814,5.440,148.592
C05107=1228.534,63.939,-45.188,-178.811,5.441,148.591
C05108=1228.529,64.189,-45.204,-178.809,5.441,148.591
C05109=1228.524,64.439,-45.221,-178.806,5.442,148.590
C05110=1228.519,64.688,-45.239,-178.804,5.443,148.589
C05111=1228.514,64.937,-45.256,-178.801,5.443,148.589
C05112=1228.509,65.186,-45.273,-178.798,5.444,148.588
C05113=1228.505,65.435,-45.290,-178.796,5.445,148.588
C05114=1228.499,65.685,-45.308,-178.794,5.445,148.587
C05115=1228.495,65.935,-45.324,-178.791,5.446,148.586
C05116=1228.490,66.184,-45.342,-178.788,5.446,148.586
C05117=1228.485,66.434,-45.360,-178.786,5.447,148.585
C05118=1228.481,66.682,-45.377,-178.783,5.448,148.584
C05119=1228.475,66.932,-45.394,-178.781,5.449,148.584
C05120=1228.470,67.181,-45.411,-178.778,5.449,148.583
C05121=1228.465,67.430,-45.429,-178.776,5.450,148.582
C05122=1228.460,67.680,-45.446,-178.773,5.450,148.582
C05123=1228.455,67.929,-45.464,-178.771,5.451,148.581
C05124=1228.451,68.179,-45.480,-178.768,5.452,148.580
C05125=1228.446,68.428,-45.498,-178.766,5.452,148.580
C05126=1228.441,68.678,-45.516,-178.763,5.453,148.579
C05127=1228.436,68.927,-45.532,-178.761,5.454,148.579
C05128=1228.431,69.176,-45.550,-178.758,5.454,148.578
C05129=1228.426,69.426,-45.568,-178.755,5.455,148.577
C05130=1228.421,69.674,-45.585,-178.753,5.456,148.577
C05131=1228.416,69.924,-45.602,-178.750,5.456,148.576
C05132=1228.411,70.173,-45.620,-178.748,5.457,148.576
C05133=1228.407,70.423,-45.637,-178.745,5.457,148.575
C05134=1228.402,70.672,-45.654,-178.743,5.458,148.574
C05135=1228.397,70.922,-45.672,-178.740,5.459,148.574
C05136=1228.392,71.171,-45.690,-178.738,5.460,148.573
C05137=1228.387,71.420,-45.707,-178.735,5.460,148.573
C05138=1228.382,71.669,-45.724,-178.733,5.461,148.572
C05139=1228.377,71.919,-45.742,-178.730,5.461,148.571
C05140=1228.373,72.168,-45.759,-178.727,5.462,148.571
C05141=1228.368,72.417,-45.777,-178.725,5.463,148.570
C05142=1228.363,72.667,-45.794,-178.723,5.463,148.569
C05143=1228.358,72.916,-45.812,-178.720,5.464,148.569
C05144=1228.353,73.165,-45.830,-178.717,5.465,148.568
C05145=1228.348,73.415,-45.847,-178.715,5.465,148.568
C05146=1228.344,73.664,-45.865,-178.713,5.466,148.567
C05147=1228.338,73.914,-45.882,-178.710,5.467,148.566
C05148=1228.333,74.163,-45.900,-178.707,5.467,148.566
C05149=1228.328,74.412,-45.918,-178.705,5.468,148.565
C05150=1228.324,74.662,-45.935,-178.702,5.469,148.564
C05151=1228.319,74.911,-45.953,-178.700,5.469,148.564
C05152=1228.314,75.160,-45.971,-178.697,5.470,148.563
C05153=1228.309,75.410,-45.988,-178.695,5.471,148.563
C05154=1228.304,75.659,-46.006,-178.692,5.471,148.562
C05155=1228.299,75.908,-46.024,-178.690,5.472,148.562
C05156=1228.295,76.157,-46.041,-178.687,5.473,148.561
C05157=1228.290,76.407,-46.059,-178.684,5.474,148.560
C05158=1228.285,76.656,-46.077,-178.681,5.475,148.560
C05159=1228.280,76.905,-46.095,-178.679,5.475,148.559
C05160=1228.275,77.155,-46.112,-178.677,5.476,148.559
C05161=1228.270,77.404,-46.130,-178.674,5.477,148.558
C05162=1228.265,77.653,-46.148,-178.671,5.478,148.557
C05163=1228.261,77.902,-46.165,-178.669,5.478,148.557
C05164=1228.256,78.151,-46.183,-178.666,5.479,148.556
C05165=1228.251,78.401,-46.200,-178.664,5.480,148.555
C05166=1228.246,78.650,-46.218,-178.661,5.480,148.555
C05167=1228.241,78.900,-46.236,-178.659,5.481,148.554
C05168=1228.236,79.149,-46.255,-178.656,5.481,148.554
C05169=1228.232,79.399,-46.273,-178.654,5.482,148.553
C05170=1228.226,79.648,-46.290,-178.651,5.483,148.552
C05171=1228.221,79.898,-46.308,-178.649,5.484,148.552
C05172=1228.216,80.147,-46.326,-178.646,5.484,148.551
C05173=1228.212,80.396,-46.344,-178.644,5.485,148.551
C05174=1228.207,80.645,-46.362,-178.641,5.486,148.550
C05175=1228.202,80.894,-46.380,-178.638,5.487,148.549
C05176=1228.197,81.144,-46.398,-178.636,5.488,148.549
C05177=1228.191,81.412,-46.417,-178.633,5.488,148.548
C05178=1228.186,81.681,-46.436,-178.630,5.489,148.547
C05179=1228.181,81.949,-46.455,-178.628,5.489,148.547
C05180=1228.176,82.217,-46.475,-178.625,5.491,148.546
C05181=1228.171,82.466,-46.493,-178.622,5.492,148.546
C05182=1228.166,82.715,-46.511,-178.620,5.492,148.545
C05183=1228.161,82.965,-46.529,-178.617,5.493,148.544
C05184=1228.157,83.215,-46.547,-178.614,5.494,148.544
C05185=1228.152,83.464,-46.565,-178.612,5.495,148.543
C05186=1228.147,83.713,-46.583,-178.610,5.495,148.543
C05187=1228.142,83.962,-46.601,-178.607,5.496,148.542
C05188=1228.138,84.211,-46.619,-178.604,5.496,148.541
C05189=1228.133,84.460,-46.637,-178.602,5.497,148.541
C05190=1228.128,84.710,-46.655,-178.600,5.498,148.540
C05191=1228.123,84.959,-46.673,-178.597,5.499,148.540
C05192=1228.118,85.209,-46.691,-178.594,5.500,148.539
C05193=1228.113,85.458,-46.710,-178.592,5.501,148.539
C05194=1228.108,85.707,-46.728,-178.589,5.502,148.538
C05195=1228.103,85.956,-46.746,-178.587,5.502,148.537
C05196=1228.099,86.206,-46.764,-178.584,5.503,148.537
C05197=1228.094,86.456,-46.782,-178.582,5.504,148.536
C05198=1228.089,86.705,-46.800,-178.579,5.504,148.535
C05199=1228.084,86.954,-46.818,-178.577,5.505,148.535
C05200=1228.079,87.203,-46.836,-178.574,5.505,148.534
C05201=1228.075,87.453,-46.854,-178.572,5.506,148.534
C05202=1228.070,87.702,-46.872,-178.569,5.508,148.533
C05203=1228.064,87.952,-46.891,-178.566,5.508,148.532
C05204=1228.060,88.200,-46.910,-178.563,5.509,148.532
C05205=1228.055,88.449,-46.928,-178.561,5.510,148.531
C05206=1228.050,88.699,-46.946,-178.559,5.511,148.531
C05207=1228.045,88.948,-46.964,-178.556,5.511,148.530
C05208=1228.041,89.198,-46.982,-178.553,5.512,148.529
C05209=1228.035,89.447,-47.001,-178.551,5.513,148.529
C05210=1228.030,89.696,-47.019,-178.549,5.513,148.528
C05211=1228.026,89.945,-47.038,-178.545,5.515,148.528
C05212=1228.021,90.195,-47.056,-178.543,5.516,148.527
C05213=1228.016,90.444,-47.074,-178.541,5.516,148.527
C05214=1228.011,90.693,-47.092,-178.538,5.517,148.526
C05215=1228.006,90.943,-47.111,-178.535,5.518,148.525
C05216=1228.002,91.192,-47.129,-178.533,5.518,148.525
C05217=1227.997,91.441,-47.147,-178.531,5.519,148.524
C05218=1227.992,91.691,-47.165,-178.528,5.520,148.524
C05219=1227.987,91.940,-47.185,-178.526,5.521,148.523
C05220=1227.982,92.189,-47.203,-178.523,5.522,148.523
C05221=1227.977,92.438,-47.221,-178.520,5.523,148.522
C05222=1227.973,92.688,-47.239,-178.518,5.523,148.521
C05223=1227.968,92.937,-47.258,-178.515,5.524,148.521
C05224=1227.963,93.186,-47.276,-178.513,5.525,148.520
C05225=1227.958,93.436,-47.295,-178.510,5.525,148.520
C05226=1227.954,93.684,-47.313,-178.508,5.526,148.519
C05227=1227.948,93.934,-47.332,-178.505,5.528,148.518
C05228=1227.943,94.183,-47.350,-178.502,5.528,148.518
C05229=1227.939,94.432,-47.369,-178.500,5.529,148.517
C05230=1227.933,94.682,-47.388,-178.497,5.530,148.517
C05231=1227.929,94.931,-47.406,-178.495,5.531,148.516
C05232=1227.925,95.180,-47.425,-178.492,5.531,148.515
C05233=1227.920,95.429,-47.443,-178.490,5.532,148.515
C05234=1227.914,95.678,-47.462,-178.487,5.534,148.514
C05235=1227.910,95.928,-47.480,-178.484,5.534,148.514
C05236=1227.905,96.177,-47.498,-178.482,5.535,148.513
C05237=1227.900,96.426,-47.517,-178.480,5.536,148.513
C05238=1227.895,96.676,-47.536,-178.477,5.536,148.512
C05239=1227.890,96.925,-47.555,-178.474,5.537,148.511
C05240=1227.885,97.174,-47.573,-178.472,5.538,148.511
C05241=1227.881,97.423,-47.592,-178.469,5.539,148.510
C05242=1227.875,97.673,-47.611,-178.466,5.540,148.510
C05243=1227.871,97.921,-47.629,-178.464,5.541,148.509
C05244=1227.867,98.171,-47.648,-178.462,5.542,148.509
C05245=1227.861,98.420,-47.667,-178.459,5.542,148.508
C05246=1227.857,98.670,-47.685,-178.457,5.543,148.508
C05247=1227.852,98.919,-47.705,-178.454,5.545,148.507
C05248=1227.847,99.168,-47.723,-178.451,5.545,148.506
C05249=1227.843,99.417,-47.742,-178.449,5.546,148.506
C05250=1227.837,99.667,-47.760,-178.446,5.547,148.505
C05251=1227.833,99.916,-47.779,-178.444,5.547,148.505
C05252=1227.827,100.166,-47.798,-178.442,5.548,148.504
C05253=1227.823,100.414,-47.817,-178.438,5.550,148.503
C05254=1227.818,100.664,-47.836,-178.436,5.550,148.503
C05255=1227.813,100.913,-47.854,-178.433,5.551,148.502
C05256=1227.809,101.162,-47.873,-178.431,5.552,148.502
C05257=1227.803,101.412,-47.892,-178.428,5.553,148.501
C05258=1227.799,101.660,-47.911,-178.426,5.553,148.500
C05259=1227.794,101.910,-47.930,-178.423,5.555,148.500
C05260=1227.789,102.159,-47.948,-178.421,5.556,148.499
C05261=1227.784,102.408,-47.968,-178.418,5.556,148.499
C05262=1227.780,102.658,-47.986,-178.416,5.557,148.498
C05263=1227.775,102.907,-48.006,-178.413,5.558,148.498
C05264=1227.770,103.156,-48.024,-178.410,5.559,148.497
C05265=1227.765,103.406,-48.043,-178.408,5.560,148.497
C05266=1227.761,103.655,-48.062,-178.405,5.561,148.496
C05267=1227.755,103.903,-48.081,-178.403,5.561,148.495
C05268=1227.750,104.154,-48.100,-178.401,5.562,148.495
C05269=1227.746,104.402,-48.119,-178.398,5.563,148.494
C05270=1227.741,104.652,-48.138,-178.395,5.565,148.494
C05271=1227.736,104.900,-48.157,-178.393,5.565,148.493
C05272=1227.731,105.150,-48.176,-178.390,5.566,148.493
C05273=1227.727,105.399,-48.195,-178.388,5.567,148.492
C05274=1227.722,105.649,-48.214,-178.385,5.567,148.492
C05275=1227.717,105.897,-48.233,-178.382,5.569,148.491
C05276=1227.712,106.147,-48.252,-178.380,5.570,148.491
C05277=1227.707,106.396,-48.271,-178.377,5.571,148.490
C05278=1227.703,106.645,-48.290,-178.375,5.571,148.489
C05279=1227.697,106.894,-48.310,-178.373,5.572,148.489
C05280=1227.693,107.144,-48.329,-178.369,5.574,148.488
C05281=1227.688,107.412,-48.349,-178.367,5.574,148.488
C05282=1227.683,107.681,-48.370,-178.364,5.575,148.487
C05283=1227.677,107.949,-48.391,-178.361,5.576,148.486
C05284=1227.672,108.218,-48.411,-178.359,5.577,148.486
C05285=1227.667,108.467,-48.430,-178.356,5.578,148.485
C05286=1227.663,108.716,-48.449,-178.353,5.579,148.485
C05287=1227.658,108.966,-48.469,-178.351,5.580,148.484
C05288=1227.653,109.214,-48.488,-178.348,5.581,148.484
C05289=1227.649,109.464,-48.507,-178.346,5.581,148.483
C05290=1227.643,109.713,-48.527,-178.344,5.582,148.482
C05291=1227.639,109.962,-48.546,-178.340,5.584,148.482
C05292=1227.634,110.211,-48.565,-178.338,5.585,148.481
C05293=1227.629,110.461,-48.584,-178.336,5.585,148.481
C05294=1227.623,110.710,-48.603,-178.333,5.586,148.480
C05295=1227.619,110.959,-48.622,-178.330,5.588,148.480
C05296=1227.615,111.209,-48.642,-178.328,5.588,148.479
C05297=1227.609,111.458,-48.661,-178.325,5.589,148.478
C05298=1227.605,111.707,-48.680,-178.323,5.590,148.478
C05299=1227.600,111.956,-48.700,-178.320,5.591,148.477
C05300=1227.595,112.205,-48.719,-178.318,5.592,148.477
C05301=1227.590,112.455,-48.739,-178.315,5.593,148.476
C05302=1227.586,112.703,-48.758,-178.313,5.594,148.476
C05303=1227.581,112.953,-48.777,-178.310,5.595,148.475
C05304=1227.576,113.202,-48.797,-178.307,5.596,148.475
C05305=1227.571,113.451,-48.816,-178.305,5.597,148.474
C05306=1227.567,113.701,-48.835,-178.303,5.598,148.474
C05307=1227.562,113.949,-48.855,-178.300,5.598,148.473
C05308=1227.557,114.198,-48.875,-178.297,5.600,148.473
C05309=1227.552,114.447,-48.894,-178.295,5.601,148.472
C05310=1227.547,114.697,-48.914,-178.292,5.601,148.471
C05311=1227.543,114.946,-48.933,-178.290,5.602,148.471
C05312=1227.538,115.195,-48.952,-178.287,5.604,148.470
C05313=1227.533,115.445,-48.972,-178.285,5.605,148.470
C05314=1227.528,115.694,-48.992,-178.282,5.605,148.469
C05315=1227.523,115.943,-49.011,-178.279,5.606,148.469
C05316=1227.518,116.193,-49.030,-178.277,5.608,148.468
C05317=1227.515,116.441,-49.050,-178.274,5.608,148.468
C05318=1227.509,116.690,-49.070,-178.272,5.609,148.467
C05319=1227.504,116.940,-49.089,-178.269,5.610,148.466
C05320=1227.500,117.189,-49.109,-178.266,5.611,148.466
C05321=1227.494,117.438,-49.128,-178.264,5.612,148.465
C05322=1227.490,117.688,-49.148,-178.261,5.613,148.465
C05323=1227.485,117.937,-49.168,-178.259,5.615,148.464
C05324=1227.481,118.185,-49.187,-178.256,5.615,148.464
C05325=1227.476,118.435,-49.207,-178.254,5.616,148.463
C05326=1227.471,118.684,-49.226,-178.251,5.617,148.463
C05327=1227.466,118.933,-49.246,-178.248,5.619,148.462
C05328=1227.461,119.182,-49.266,-178.246,5.619,148.462
C05329=1227.457,119.432,-49.285,-178.244,5.620,148.461
C05330=1227.452,119.681,-49.305,-178.241,5.621,148.461
C05331=1227.447,119.929,-49.325,-178.238,5.623,148.460
C05332=1227.442,120.179,-49.345,-178.236,5.623,148.459
C05333=1227.437,120.429,-49.364,-178.234,5.624,148.459
C05334=1227.432,120.677,-49.384,-178.230,5.626,148.458
C05335=1227.428,120.926,-49.404,-178.228,5.627,148.458
C05336=1227.423,121.176,-49.424,-178.226,5.627,148.457
C05337=1227.418,121.426,-49.443,-178.224,5.628,148.457
C05338=1227.413,121.674,-49.463,-178.220,5.630,148.456
C05339=1227.408,121.923,-49.483,-178.218,5.630,148.456
C05340=1227.404,122.172,-49.503,-178.216,5.631,148.455
C05341=1227.399,122.422,-49.523,-178.212,5.633,148.455
C05342=1227.394,122.671,-49.542,-178.210,5.634,148.454
C05343=1227.389,122.920,-49.563,-178.208,5.634,148.454
C05344=1227.385,123.169,-49.582,-178.206,5.635,148.453
C05345=1227.380,123.419,-49.602,-178.202,5.637,148.453
C05346=1227.375,123.668,-49.622,-178.200,5.638,148.452
C05347=1227.370,123.917,-49.642,-178.198,5.638,148.451
C05348=1227.366,124.166,-49.662,-178.195,5.640,148.451
C05349=1227.361,124.415,-49.682,-178.192,5.641,148.450
C05350=1227.356,124.664,-49.702,-178.190,5.641,148.450
C05351=1227.351,124.913,-49.721,-178.187,5.643,148.449
C05352=1227.347,125.162,-49.742,-178.185,5.644,148.449
C05353=1227.342,125.412,-49.761,-178.182,5.645,148.448
C05354=1227.337,125.660,-49.782,-178.179,5.646,148.448
C05355=1227.333,125.910,-49.802,-178.177,5.647,148.447
C05356=1227.328,126.159,-49.822,-178.175,5.648,148.447
C05357=1227.323,126.408,-49.841,-178.172,5.648,148.446
C05358=1227.319,126.657,-49.862,-178.169,5.650,148.446
C05359=1227.313,126.907,-49.882,-178.167,5.651,148.445
C05360=1227.309,127.156,-49.902,-178.165,5.652,148.445
C05361=1227.304,127.405,-49.922,-178.161,5.653,148.444
C05362=1227.299,127.654,-49.942,-178.159,5.654,148.444
C05363=1227.294,127.903,-49.961,-178.157,5.655,148.443
C05364=1227.290,128.152,-49.982,-178.154,5.657,148.443
C05365=1227.285,128.401,-50.002,-178.151,5.657,148.442
C05366=1227.280,128.650,-50.022,-178.149,5.658,148.442
C05367=1227.275,128.900,-50.043,-178.146,5.660,148.441
C05368=1227.271,129.149,-50.063,-178.144,5.661,148.441
C05369=1227.266,129.398,-50.083,-178.141,5.661,148.440
C05370=1227.261,129.647,-50.103,-178.139,5.663,148.440
C05371=1227.256,129.896,-50.123,-178.136,5.664,148.439
C05372=1227.252,130.145,-50.143,-178.133,5.664,148.438
C05373=1227.247,130.394,-50.164,-178.131,5.666,148.438
C05374=1227.242,130.644,-50.184,-178.128,5.667,148.437
C05375=1227.238,130.893,-50.204,-178.126,5.668,148.437
C05376=1227.233,131.142,-50.224,-178.123,5.669,148.436
C05377=1227.228,131.392,-50.245,-178.121,5.670,148.436
C05378=1227.223,131.641,-50.265,-178.118,5.671,148.435
C05379=1227.218,131.889,-50.285,-178.116,5.673,148.435
C05380=1227.214,132.138,-50.305,-178.113,5.673,148.434
C05381=1227.208,132.388,-50.326,-178.111,5.674,148.434
C05382=1227.204,132.637,-50.346,-178.108,5.676,148.433
C05383=1227.199,132.886,-50.366,-178.106,5.677,148.433
C05384=1227.195,133.135,-50.387,-178.102,5.678,148.432
C05385=1227.189,133.403,-50.408,-178.100,5.679,148.432
C05386=1227.185,133.673,-50.431,-178.097,5.681,148.431
C05387=1227.180,133.941,-50.452,-178.094,5.681,148.431
C05388=1227.174,134.210,-50.475,-178.091,5.683,148.430
C05389=1227.170,134.458,-50.495,-178.089,5.684,148.429
C05390=1227.165,134.708,-50.516,-178.087,5.684,148.429
C05391=1227.160,134.957,-50.536,-178.084,5.686,148.428
C05392=1227.155,135.206,-50.556,-178.081,5.687,148.428
C05393=1227.150,135.456,-50.577,-178.079,5.689,148.427
C05394=1227.146,135.704,-50.597,-178.076,5.689,148.427
C05395=1227.141,135.953,-50.618,-178.074,5.690,148.426
C05396=1227.136,136.203,-50.639,-178.071,5.692,148.426
C05397=1227.132,136.452,-50.659,-178.069,5.693,148.425
C05398=1227.127,136.701,-50.679,-178.067,5.694,148.425
C05399=1227.122,136.950,-50.700,-178.063,5.695,148.424
C05400=1227.117,137.199,-50.720,-178.061,5.696,148.424
C05401=1227.112,137.449,-50.741,-178.058,5.698,148.423
C05402=1227.108,137.698,-50.761,-178.056,5.699,148.423
C05403=1227.103,137.947,-50.782,-178.053,5.699,148.422
C05404=1227.098,138.196,-50.803,-178.051,5.701,148.422
C05405=1227.094,138.445,-50.823,-178.048,5.702,148.421
C05406=1227.089,138.694,-50.844,-178.046,5.703,148.421
C05407=1227.084,138.943,-50.864,-178.043,5.704,148.420
C05408=1227.080,139.192,-50.885,-178.041,5.705,148.420
C05409=1227.075,139.441,-50.906,-178.038,5.707,148.419
C05410=1227.070,139.690,-50.926,-178.036,5.708,148.419
C05411=1227.065,139.939,-50.947,-178.033,5.708,148.418
C05412=1227.061,140.188,-50.967,-178.030,5.710,148.418
C05413=1227.055,140.438,-50.988,-178.028,5.711,148.417
C05414=1227.051,140.687,-51.009,-178.025,5.713,148.417
C05415=1227.046,140.936,-51.030,-178.022,5.713,148.416
C05416=1227.042,141.184,-51.051,-178.020,5.714,148.416
C05417=1227.036,141.433,-51.072,-178.018,5.716,148.416
C05418=1227.032,141.682,-51.092,-178.015,5.717,148.415
C05419=1227.027,141.932,-51.113,-178.012,5.718,148.415
C05420=1227.023,142.181,-51.134,-178.010,5.719,148.414
C05421=1227.018,142.431,-51.155,-178.008,5.720,148.413
C05422=1227.013,142.679,-51.175,-178.004,5.722,148.413
C05423=1227.008,142.929,-51.196,-178.002,5.723,148.412
C05424=1227.004,143.177,-51.217,-177.999,5.724,148.412
C05425=1226.999,143.426,-51.238,-177.997,5.725,148.411
C05426=1226.994,143.675,-51.259,-177.994,5.726,148.411
C05427=1226.989,143.924,-51.280,-177.992,5.727,148.410
C05428=1226.985,144.173,-51.300,-177.990,5.728,148.410
C05429=1226.980,144.423,-51.321,-177.987,5.730,148.409
C05430=1226.976,144.672,-51.342,-177.984,5.731,148.409
C05431=1226.971,144.921,-51.363,-177.981,5.732,148.408
C05432=1226.966,145.170,-51.384,-177.979,5.733,148.408
C05433=1226.961,145.419,-51.405,-177.977,5.734,148.407
C05434=1226.956,145.668,-51.426,-177.974,5.736,148.407
C05435=1226.952,145.917,-51.447,-177.971,5.736,148.406
C05436=1226.947,146.166,-51.468,-177.969,5.738,148.406
C05437=1226.942,146.416,-51.489,-177.967,5.739,148.406
C05438=1226.938,146.664,-51.510,-177.963,5.741,148.405
C05439=1226.933,146.914,-51.531,-177.961,5.742,148.405
C05440=1226.928,147.163,-51.552,-177.959,5.742,148.404
C05441=1226.924,147.411,-51.573,-177.956,5.744,148.404
C05442=1226.918,147.660,-51.594,-177.953,5.745,148.403
C05443=1226.915,147.910,-51.615,-177.951,5.747,148.403
C05444=1226.910,148.159,-51.637,-177.949,5.748,148.402
C05445=1226.905,148.408,-51.657,-177.945,5.749,148.402
C05446=1226.900,148.657,-51.678,-177.943,5.750,148.401
C05447=1226.895,148.906,-51.700,-177.940,5.752,148.401
C05448=1226.891,149.156,-51.721,-177.938,5.753,148.400
C05449=1226.886,149.404,-51.743,-177.936,5.754,148.400
C05450=1226.881,149.653,-51.763,-177.933,5.755,148.399
C05451=1226.876,149.902,-51.784,-177.931,5.756,148.399
C05452=1226.871,150.151,-51.806,-177.928,5.757,148.398
C05453=1226.868,150.401,-51.826,-177.926,5.758,148.398
C05454=1226.863,150.649,-51.848,-177.922,5.760,148.397
C05455=1226.857,150.899,-51.869,-177.920,5.761,148.397
C05456=1226.853,151.147,-51.891,-177.918,5.763,148.397
C05457=1226.848,151.396,-51.911,-177.915,5.763,148.396
C05458=1226.844,151.646,-51.933,-177.912,5.765,148.396
C05459=1226.839,151.895,-51.954,-177.910,5.766,148.395
C05460=1226.834,152.143,-51.976,-177.907,5.768,148.395
C05461=1226.829,152.392,-51.996,-177.905,5.769,148.394
C05462=1226.825,152.642,-52.018,-177.902,5.769,148.393
C05463=1226.820,152.891,-52.039,-177.900,5.771,148.393
C05464=1226.815,153.140,-52.061,-177.897,5.772,148.392
C05465=1226.810,153.389,-52.082,-177.894,5.774,148.392
C05466=1226.806,153.638,-52.103,-177.892,5.775,148.392
C05467=1226.801,153.887,-52.124,-177.889,5.776,148.391
C05468=1226.796,154.136,-52.146,-177.887,5.777,148.391
C05469=1226.792,154.385,-52.168,-177.884,5.779,148.390
C05470=1226.787,154.634,-52.189,-177.882,5.780,148.390
C05471=1226.782,154.883,-52.211,-177.879,5.781,148.389
C05472=1226.778,155.132,-52.231,-177.877,5.782,148.389
C05473=1226.773,155.381,-52.253,-177.874,5.784,148.388
C05474=1226.768,155.630,-52.275,-177.872,5.785,148.388
C05475=1226.763,155.879,-52.296,-177.869,5.786,148.387
C05476=1226.759,156.129,-52.318,-177.867,5.787,148.387
C05477=1226.754,156.377,-52.339,-177.864,5.789,148.387
C05478=1226.749,156.626,-52.360,-177.861,5.790,148.386
C05479=1226.745,156.876,-52.382,-177.859,5.792,148.386
C05480=1226.740,157.124,-52.404,-177.856,5.792,148.385
